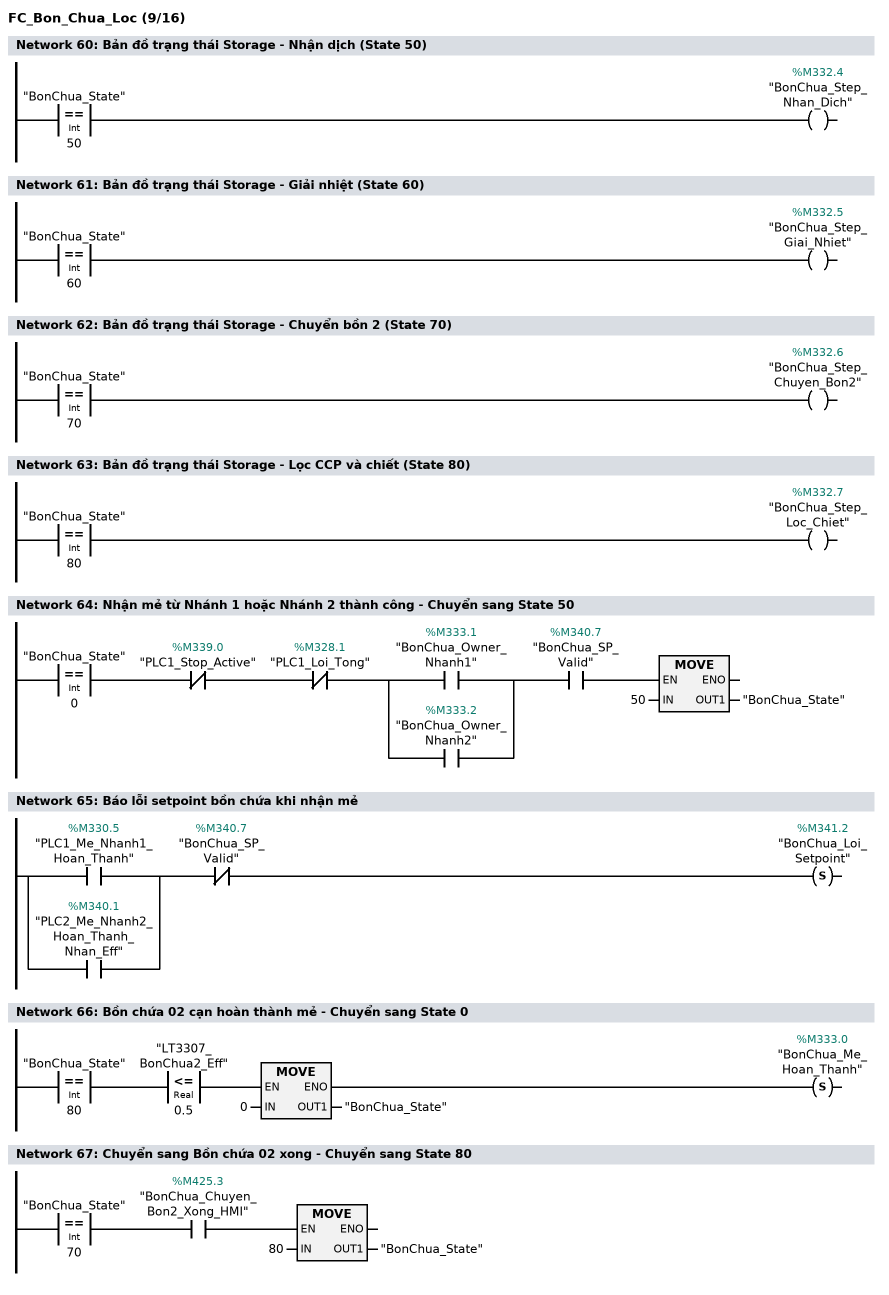
   RUNG wire#powerrail
      { S7_Templates := "SrcType := Int" } EQ_Contact(in1 := "BonChua_State", in2 := 50)
      Coil( "BonChua_Step_Nhan_Dich" )
   END_RUNG
   // the same network as SCL:
   "BonChua_Step_Nhan_Dich" := "BonChua_State" = 50;
END_REGION

REGION Network 61: Bản đồ trạng thái Storage - Giải nhiệt (State 60)
   RUNG wire#powerrail
      { S7_Templates := "SrcType := Int" } EQ_Contact(in1 := "BonChua_State", in2 := 60)
      Coil( "BonChua_Step_Giai_Nhiet" )
   END_RUNG
   // the same network as SCL:
   "BonChua_Step_Giai_Nhiet" := "BonChua_State" = 60;
END_REGION

REGION Network 62: Bản đồ trạng thái Storage - Chuyển bồn 2 (State 70)
   RUNG wire#powerrail
      { S7_Templates := "SrcType := Int" } EQ_Contact(in1 := "BonChua_State", in2 := 70)
      Coil( "BonChua_Step_Chuyen_Bon2" )
   END_RUNG
   // the same network as SCL:
   "BonChua_Step_Chuyen_Bon2" := "BonChua_State" = 70;
END_REGION

REGION Network 63: Bản đồ trạng thái Storage - Lọc CCP và chiết (State 80)
   RUNG wire#powerrail
      { S7_Templates := "SrcType := Int" } EQ_Contact(in1 := "BonChua_State", in2 := 80)
      Coil( "BonChua_Step_Loc_Chiet" )
   END_RUNG
   // the same network as SCL:
   "BonChua_Step_Loc_Chiet" := "BonChua_State" = 80;
END_REGION

REGION Network 64: Nhận mẻ từ Nhánh 1 hoặc Nhánh 2 thành công - Chuyển sang State 50
   RUNG wire#powerrail
      { S7_Templates := "SrcType := Int" } EQ_Contact(in1 := "BonChua_State", in2 := 0)
      I_Contact( "PLC1_Stop_Active" )
      I_Contact( "PLC1_Loi_Tong" )
      wire#w1
      Contact( "BonChua_Owner_Nhanh1" )
      wire#w2
      Contact( "BonChua_SP_Valid" )
      { S7_GenerateENO := "TRUE" } Move(in := 50, out1 => "BonChua_State")
   END_RUNG
   RUNG wire#w1
      Contact( "BonChua_Owner_Nhanh2" )
   END_RUNG wire#w2
   // the same network as SCL:
   IF ("BonChua_State" = 0) AND NOT "PLC1_Stop_Active" AND NOT "PLC1_Loi_Tong" AND ("BonChua_Owner_Nhanh1" OR "BonChua_Owner_Nhanh2") AND "BonChua_SP_Valid" THEN
       "BonChua_State" := 50;
   END_IF;
END_REGION

REGION Network 65: Báo lỗi setpoint bồn chứa khi nhận mẻ
   RUNG wire#powerrail
      Contact( "PLC1_Me_Nhanh1_Hoan_Thanh" )
      wire#w1
      I_Contact( "BonChua_SP_Valid" )
      S_Coil( "BonChua_Loi_Setpoint" )
   END_RUNG
   RUNG wire#powerrail
      Contact( "PLC2_Me_Nhanh2_Hoan_Thanh_Nhan_Eff" )
   END_RUNG wire#w1
   // the same network as SCL:
   IF ("PLC1_Me_Nhanh1_Hoan_Thanh" OR "PLC2_Me_Nhanh2_Hoan_Thanh_Nhan_Eff") AND NOT "BonChua_SP_Valid" THEN
       "BonChua_Loi_Setpoint" := TRUE;
   END_IF;
END_REGION

REGION Network 66: Bồn chứa 02 cạn hoàn thành mẻ - Chuyển sang State 0
   RUNG wire#powerrail
      { S7_Templates := "SrcType := Int" } EQ_Contact(in1 := "BonChua_State", in2 := 80)
      { S7_Templates := "SrcType := Real" } LE_Contact(in1 := "LT3307_BonChua2_Eff", in2 := 0.5)
      { S7_GenerateENO := "TRUE" } Move(in := 0, out1 => "BonChua_State")
      S_Coil( "BonChua_Me_Hoan_Thanh" )
   END_RUNG
   // the same network as SCL:
   // ENO of a box is taken as its EN; it also drops when the box reports an error
   #_w1 := ("BonChua_State" = 80) AND ("LT3307_BonChua2_Eff" <= 0.5);
   IF #_w1 THEN
       "BonChua_State" := 0;
       "BonChua_Me_Hoan_Thanh" := TRUE;
   END_IF;
END_REGION

REGION Network 67: Chuyển sang Bồn chứa 02 xong - Chuyển sang State 80
   RUNG wire#powerrail
      { S7_Templates := "SrcType := Int" } EQ_Contact(in1 := "BonChua_State", in2 := 70)
      Contact( "BonChua_Chuyen_Bon2_Xong_HMI" )
      { S7_GenerateENO := "TRUE" } Move(in := 80, out1 => "BonChua_State")
   END_RUNG
   // the same network as SCL:
   IF ("BonChua_State" = 70) AND "BonChua_Chuyen_Bon2_Xong_HMI" THEN "BonChua_State" := 80; END_IF;
END_REGION

REGION Network 68: Đạt 45 độ C chuyển Bồn chứa 02 - Chuyển sang State 70
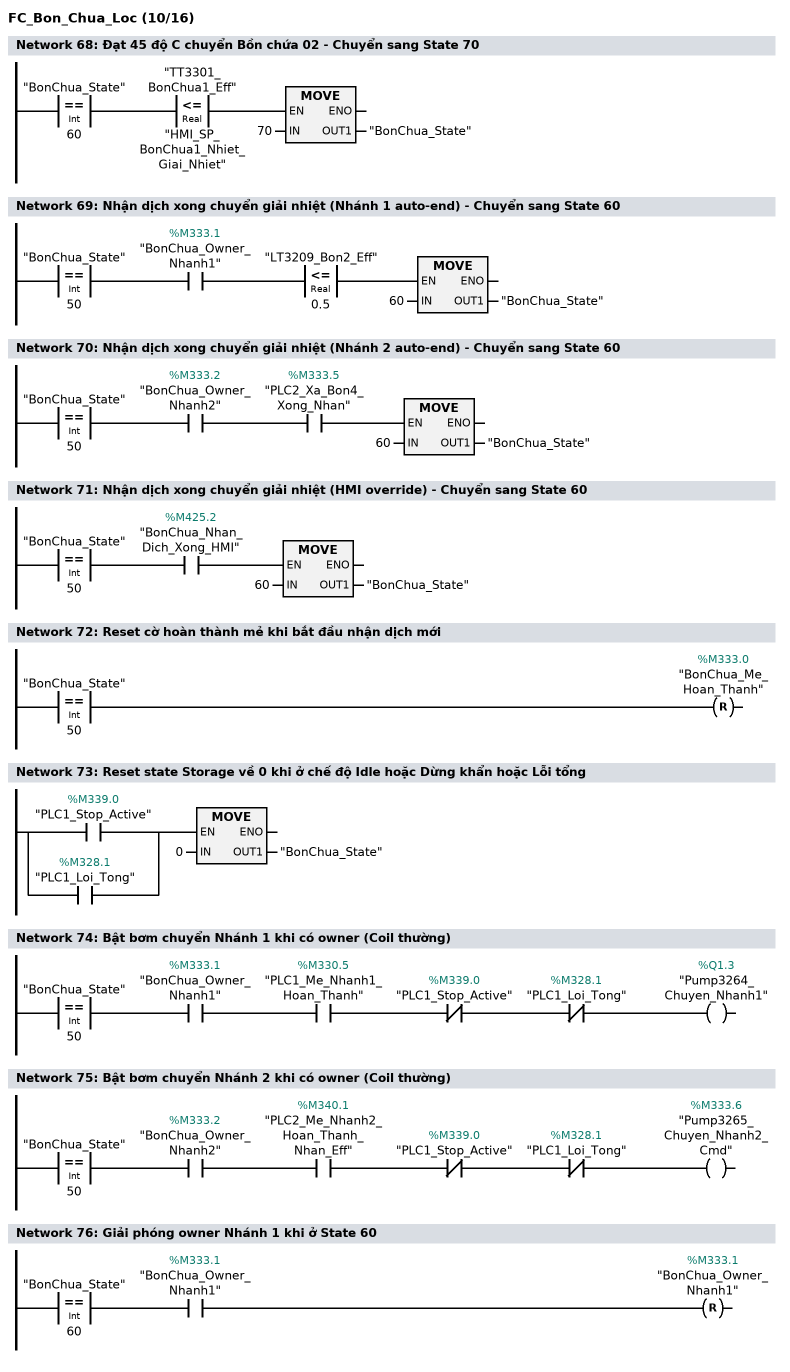
   RUNG wire#powerrail
      { S7_Templates := "SrcType := Int" } EQ_Contact(in1 := "BonChua_State", in2 := 60)
      { S7_Templates := "SrcType := Real" } LE_Contact(in1 := "TT3301_BonChua1_Eff", in2 := "HMI_SP_BonChua1_Nhiet_Giai_Nhiet")
      { S7_GenerateENO := "TRUE" } Move(in := 70, out1 => "BonChua_State")
   END_RUNG
   // the same network as SCL:
   IF ("BonChua_State" = 60) AND ("TT3301_BonChua1_Eff" <= "HMI_SP_BonChua1_Nhiet_Giai_Nhiet") THEN
       "BonChua_State" := 70;
   END_IF;
END_REGION

REGION Network 69: Nhận dịch xong chuyển giải nhiệt (Nhánh 1 auto-end) - Chuyển sang State 60
   RUNG wire#powerrail
      { S7_Templates := "SrcType := Int" } EQ_Contact(in1 := "BonChua_State", in2 := 50)
      Contact( "BonChua_Owner_Nhanh1" )
      { S7_Templates := "SrcType := Real" } LE_Contact(in1 := "LT3209_Bon2_Eff", in2 := 0.5)
      { S7_GenerateENO := "TRUE" } Move(in := 60, out1 => "BonChua_State")
   END_RUNG
   // the same network as SCL:
   IF ("BonChua_State" = 50) AND "BonChua_Owner_Nhanh1" AND ("LT3209_Bon2_Eff" <= 0.5) THEN
       "BonChua_State" := 60;
   END_IF;
END_REGION

REGION Network 70: Nhận dịch xong chuyển giải nhiệt (Nhánh 2 auto-end) - Chuyển sang State 60
   RUNG wire#powerrail
      { S7_Templates := "SrcType := Int" } EQ_Contact(in1 := "BonChua_State", in2 := 50)
      Contact( "BonChua_Owner_Nhanh2" )
      Contact( "PLC2_Xa_Bon4_Xong_Nhan" )
      { S7_GenerateENO := "TRUE" } Move(in := 60, out1 => "BonChua_State")
   END_RUNG
   // the same network as SCL:
   IF ("BonChua_State" = 50) AND "BonChua_Owner_Nhanh2" AND "PLC2_Xa_Bon4_Xong_Nhan" THEN
       "BonChua_State" := 60;
   END_IF;
END_REGION

REGION Network 71: Nhận dịch xong chuyển giải nhiệt (HMI override) - Chuyển sang State 60
   RUNG wire#powerrail
      { S7_Templates := "SrcType := Int" } EQ_Contact(in1 := "BonChua_State", in2 := 50)
      Contact( "BonChua_Nhan_Dich_Xong_HMI" )
      { S7_GenerateENO := "TRUE" } Move(in := 60, out1 => "BonChua_State")
   END_RUNG
   // the same network as SCL:
   IF ("BonChua_State" = 50) AND "BonChua_Nhan_Dich_Xong_HMI" THEN "BonChua_State" := 60; END_IF;
END_REGION

REGION Network 72: Reset cờ hoàn thành mẻ khi bắt đầu nhận dịch mới
   RUNG wire#powerrail
      { S7_Templates := "SrcType := Int" } EQ_Contact(in1 := "BonChua_State", in2 := 50)
      R_Coil( "BonChua_Me_Hoan_Thanh" )
   END_RUNG
   // the same network as SCL:
   IF "BonChua_State" = 50 THEN "BonChua_Me_Hoan_Thanh" := FALSE; END_IF;
END_REGION

REGION Network 73: Reset state Storage về 0 khi ở chế độ Idle hoặc Dừng khẩn hoặc Lỗi tổng
   RUNG wire#powerrail
      Contact( "PLC1_Stop_Active" )
      wire#w1
      { S7_GenerateENO := "TRUE" } Move(in := 0, out1 => "BonChua_State")
   END_RUNG
   RUNG wire#powerrail
      Contact( "PLC1_Loi_Tong" )
   END_RUNG wire#w1
   // the same network as SCL:
   IF "PLC1_Stop_Active" OR "PLC1_Loi_Tong" THEN "BonChua_State" := 0; END_IF;
END_REGION

REGION Network 74: Bật bơm chuyển Nhánh 1 khi có owner (Coil thường)
   RUNG wire#powerrail
      { S7_Templates := "SrcType := Int" } EQ_Contact(in1 := "BonChua_State", in2 := 50)
      Contact( "BonChua_Owner_Nhanh1" )
      Contact( "PLC1_Me_Nhanh1_Hoan_Thanh" )
      I_Contact( "PLC1_Stop_Active" )
      I_Contact( "PLC1_Loi_Tong" )
      Coil( "Pump3264_Chuyen_Nhanh1" )
   END_RUNG
   // the same network as SCL:
   "Pump3264_Chuyen_Nhanh1" := ("BonChua_State" = 50) AND "BonChua_Owner_Nhanh1" AND "PLC1_Me_Nhanh1_Hoan_Thanh" AND NOT "PLC1_Stop_Active" AND NOT "PLC1_Loi_Tong";
END_REGION

REGION Network 75: Bật bơm chuyển Nhánh 2 khi có owner (Coil thường)
   RUNG wire#powerrail
      { S7_Templates := "SrcType := Int" } EQ_Contact(in1 := "BonChua_State", in2 := 50)
      Contact( "BonChua_Owner_Nhanh2" )
      Contact( "PLC2_Me_Nhanh2_Hoan_Thanh_Nhan_Eff" )
      I_Contact( "PLC1_Stop_Active" )
      I_Contact( "PLC1_Loi_Tong" )
      Coil( "Pump3265_Chuyen_Nhanh2_Cmd" )
   END_RUNG
   // the same network as SCL:
   "Pump3265_Chuyen_Nhanh2_Cmd" := ("BonChua_State" = 50) AND "BonChua_Owner_Nhanh2" AND "PLC2_Me_Nhanh2_Hoan_Thanh_Nhan_Eff" AND NOT "PLC1_Stop_Active" AND NOT "PLC1_Loi_Tong";
END_REGION

REGION Network 76: Giải phóng owner Nhánh 1 khi ở State 60
   RUNG wire#powerrail
      { S7_Templates := "SrcType := Int" } EQ_Contact(in1 := "BonChua_State", in2 := 60)
      Contact( "BonChua_Owner_Nhanh1" )
      R_Coil( "BonChua_Owner_Nhanh1" )
   END_RUNG
   // the same network as SCL:
   IF ("BonChua_State" = 60) AND "BonChua_Owner_Nhanh1" THEN "BonChua_Owner_Nhanh1" := FALSE; END_IF;
END_REGION

REGION Network 77: Giải phóng owner Nhánh 2 khi ở State 60
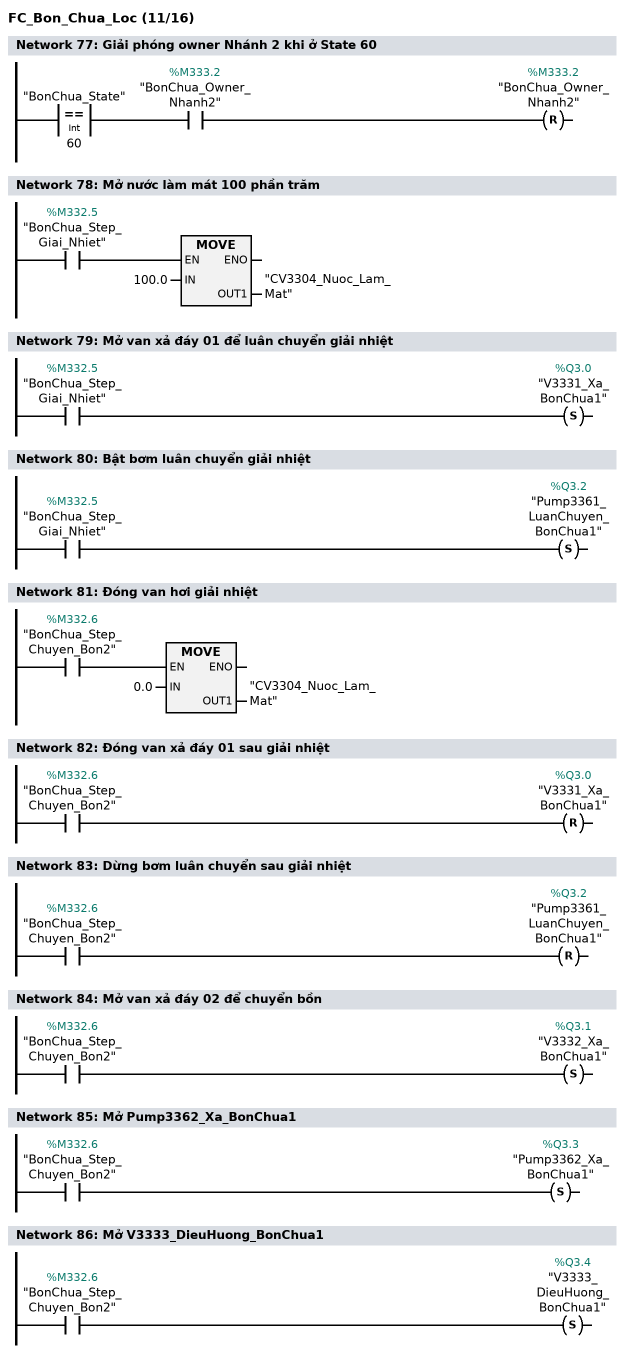
   RUNG wire#powerrail
      { S7_Templates := "SrcType := Int" } EQ_Contact(in1 := "BonChua_State", in2 := 60)
      Contact( "BonChua_Owner_Nhanh2" )
      R_Coil( "BonChua_Owner_Nhanh2" )
   END_RUNG
   // the same network as SCL:
   IF ("BonChua_State" = 60) AND "BonChua_Owner_Nhanh2" THEN "BonChua_Owner_Nhanh2" := FALSE; END_IF;
END_REGION

REGION Network 78: Mở nước làm mát 100 phần trăm
   RUNG wire#powerrail
      Contact( "BonChua_Step_Giai_Nhiet" )
      { S7_GenerateENO := "TRUE" } Move(in := 100.0, out1 => "CV3304_Nuoc_Lam_Mat")
   END_RUNG
   // the same network as SCL:
   IF "BonChua_Step_Giai_Nhiet" THEN "CV3304_Nuoc_Lam_Mat" := 100.0; END_IF;
END_REGION

REGION Network 79: Mở van xả đáy 01 để luân chuyển giải nhiệt
   RUNG wire#powerrail
      Contact( "BonChua_Step_Giai_Nhiet" )
      S_Coil( "V3331_Xa_BonChua1" )
   END_RUNG
   // the same network as SCL:
   IF "BonChua_Step_Giai_Nhiet" THEN "V3331_Xa_BonChua1" := TRUE; END_IF;
END_REGION

REGION Network 80: Bật bơm luân chuyển giải nhiệt
   RUNG wire#powerrail
      Contact( "BonChua_Step_Giai_Nhiet" )
      S_Coil( "Pump3361_LuanChuyen_BonChua1" )
   END_RUNG
   // the same network as SCL:
   IF "BonChua_Step_Giai_Nhiet" THEN "Pump3361_LuanChuyen_BonChua1" := TRUE; END_IF;
END_REGION

REGION Network 81: Đóng van hơi giải nhiệt
   RUNG wire#powerrail
      Contact( "BonChua_Step_Chuyen_Bon2" )
      { S7_GenerateENO := "TRUE" } Move(in := 0.0, out1 => "CV3304_Nuoc_Lam_Mat")
   END_RUNG
   // the same network as SCL:
   IF "BonChua_Step_Chuyen_Bon2" THEN "CV3304_Nuoc_Lam_Mat" := 0.0; END_IF;
END_REGION

REGION Network 82: Đóng van xả đáy 01 sau giải nhiệt
   RUNG wire#powerrail
      Contact( "BonChua_Step_Chuyen_Bon2" )
      R_Coil( "V3331_Xa_BonChua1" )
   END_RUNG
   // the same network as SCL:
   IF "BonChua_Step_Chuyen_Bon2" THEN "V3331_Xa_BonChua1" := FALSE; END_IF;
END_REGION

REGION Network 83: Dừng bơm luân chuyển sau giải nhiệt
   RUNG wire#powerrail
      Contact( "BonChua_Step_Chuyen_Bon2" )
      R_Coil( "Pump3361_LuanChuyen_BonChua1" )
   END_RUNG
   // the same network as SCL:
   IF "BonChua_Step_Chuyen_Bon2" THEN "Pump3361_LuanChuyen_BonChua1" := FALSE; END_IF;
END_REGION

REGION Network 84: Mở van xả đáy 02 để chuyển bồn
   RUNG wire#powerrail
      Contact( "BonChua_Step_Chuyen_Bon2" )
      S_Coil( "V3332_Xa_BonChua1" )
   END_RUNG
   // the same network as SCL:
   IF "BonChua_Step_Chuyen_Bon2" THEN "V3332_Xa_BonChua1" := TRUE; END_IF;
END_REGION

REGION Network 85: Mở Pump3362_Xa_BonChua1
   RUNG wire#powerrail
      Contact( "BonChua_Step_Chuyen_Bon2" )
      S_Coil( "Pump3362_Xa_BonChua1" )
   END_RUNG
   // the same network as SCL:
   IF "BonChua_Step_Chuyen_Bon2" THEN "Pump3362_Xa_BonChua1" := TRUE; END_IF;
END_REGION

REGION Network 86: Mở V3333_DieuHuong_BonChua1
   RUNG wire#powerrail
      Contact( "BonChua_Step_Chuyen_Bon2" )
      S_Coil( "V3333_DieuHuong_BonChua1" )
   END_RUNG
   // the same network as SCL:
   IF "BonChua_Step_Chuyen_Bon2" THEN "V3333_DieuHuong_BonChua1" := TRUE; END_IF;
END_REGION

REGION Network 87: Mở V3334_DieuHuong_BonChua1
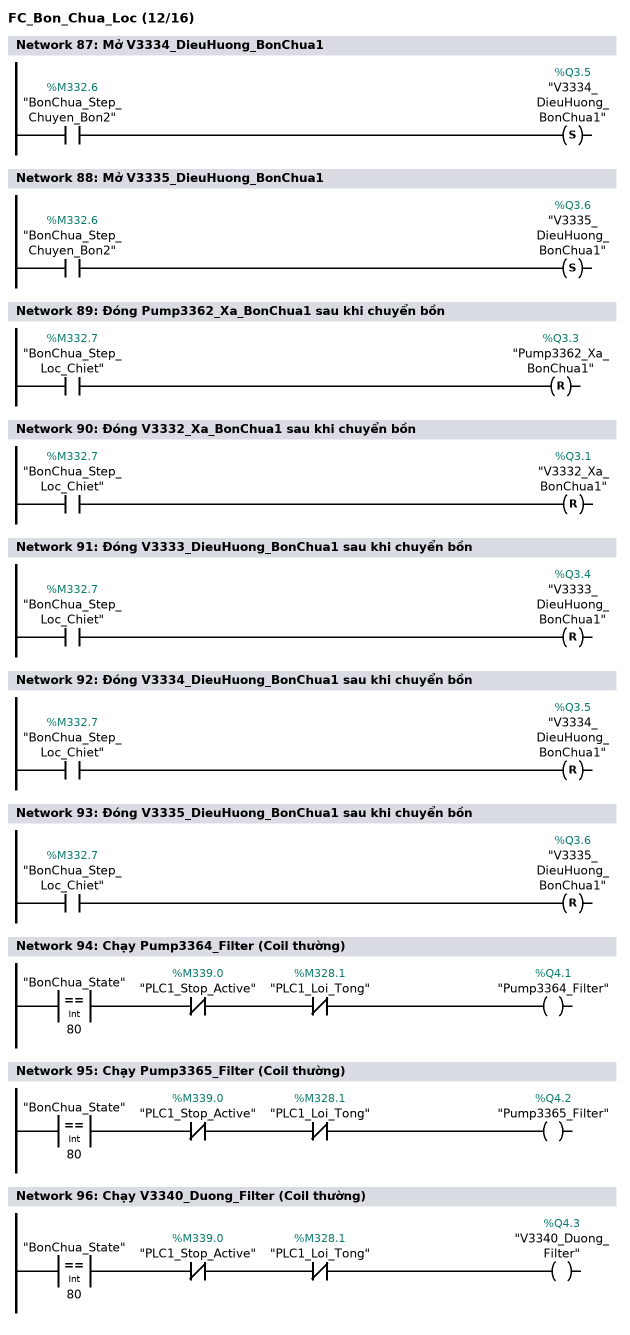
   RUNG wire#powerrail
      Contact( "BonChua_Step_Chuyen_Bon2" )
      S_Coil( "V3334_DieuHuong_BonChua1" )
   END_RUNG
   // the same network as SCL:
   IF "BonChua_Step_Chuyen_Bon2" THEN "V3334_DieuHuong_BonChua1" := TRUE; END_IF;
END_REGION

REGION Network 88: Mở V3335_DieuHuong_BonChua1
   RUNG wire#powerrail
      Contact( "BonChua_Step_Chuyen_Bon2" )
      S_Coil( "V3335_DieuHuong_BonChua1" )
   END_RUNG
   // the same network as SCL:
   IF "BonChua_Step_Chuyen_Bon2" THEN "V3335_DieuHuong_BonChua1" := TRUE; END_IF;
END_REGION

REGION Network 89: Đóng Pump3362_Xa_BonChua1 sau khi chuyển bồn
   RUNG wire#powerrail
      Contact( "BonChua_Step_Loc_Chiet" )
      R_Coil( "Pump3362_Xa_BonChua1" )
   END_RUNG
   // the same network as SCL:
   IF "BonChua_Step_Loc_Chiet" THEN "Pump3362_Xa_BonChua1" := FALSE; END_IF;
END_REGION

REGION Network 90: Đóng V3332_Xa_BonChua1 sau khi chuyển bồn
   RUNG wire#powerrail
      Contact( "BonChua_Step_Loc_Chiet" )
      R_Coil( "V3332_Xa_BonChua1" )
   END_RUNG
   // the same network as SCL:
   IF "BonChua_Step_Loc_Chiet" THEN "V3332_Xa_BonChua1" := FALSE; END_IF;
END_REGION

REGION Network 91: Đóng V3333_DieuHuong_BonChua1 sau khi chuyển bồn
   RUNG wire#powerrail
      Contact( "BonChua_Step_Loc_Chiet" )
      R_Coil( "V3333_DieuHuong_BonChua1" )
   END_RUNG
   // the same network as SCL:
   IF "BonChua_Step_Loc_Chiet" THEN "V3333_DieuHuong_BonChua1" := FALSE; END_IF;
END_REGION

REGION Network 92: Đóng V3334_DieuHuong_BonChua1 sau khi chuyển bồn
   RUNG wire#powerrail
      Contact( "BonChua_Step_Loc_Chiet" )
      R_Coil( "V3334_DieuHuong_BonChua1" )
   END_RUNG
   // the same network as SCL:
   IF "BonChua_Step_Loc_Chiet" THEN "V3334_DieuHuong_BonChua1" := FALSE; END_IF;
END_REGION

REGION Network 93: Đóng V3335_DieuHuong_BonChua1 sau khi chuyển bồn
   RUNG wire#powerrail
      Contact( "BonChua_Step_Loc_Chiet" )
      R_Coil( "V3335_DieuHuong_BonChua1" )
   END_RUNG
   // the same network as SCL:
   IF "BonChua_Step_Loc_Chiet" THEN "V3335_DieuHuong_BonChua1" := FALSE; END_IF;
END_REGION

REGION Network 94: Chạy Pump3364_Filter (Coil thường)
   RUNG wire#powerrail
      { S7_Templates := "SrcType := Int" } EQ_Contact(in1 := "BonChua_State", in2 := 80)
      I_Contact( "PLC1_Stop_Active" )
      I_Contact( "PLC1_Loi_Tong" )
      Coil( "Pump3364_Filter" )
   END_RUNG
   // the same network as SCL:
   "Pump3364_Filter" := ("BonChua_State" = 80) AND NOT "PLC1_Stop_Active" AND NOT "PLC1_Loi_Tong";
END_REGION

REGION Network 95: Chạy Pump3365_Filter (Coil thường)
   RUNG wire#powerrail
      { S7_Templates := "SrcType := Int" } EQ_Contact(in1 := "BonChua_State", in2 := 80)
      I_Contact( "PLC1_Stop_Active" )
      I_Contact( "PLC1_Loi_Tong" )
      Coil( "Pump3365_Filter" )
   END_RUNG
   // the same network as SCL:
   "Pump3365_Filter" := ("BonChua_State" = 80) AND NOT "PLC1_Stop_Active" AND NOT "PLC1_Loi_Tong";
END_REGION

REGION Network 96: Chạy V3340_Duong_Filter (Coil thường)
   RUNG wire#powerrail
      { S7_Templates := "SrcType := Int" } EQ_Contact(in1 := "BonChua_State", in2 := 80)
      I_Contact( "PLC1_Stop_Active" )
      I_Contact( "PLC1_Loi_Tong" )
      Coil( "V3340_Duong_Filter" )
   END_RUNG
   // the same network as SCL:
   "V3340_Duong_Filter" := ("BonChua_State" = 80) AND NOT "PLC1_Stop_Active" AND NOT "PLC1_Loi_Tong";
END_REGION

REGION Network 97: Chạy V3341_Duong_Filter (Coil thường)
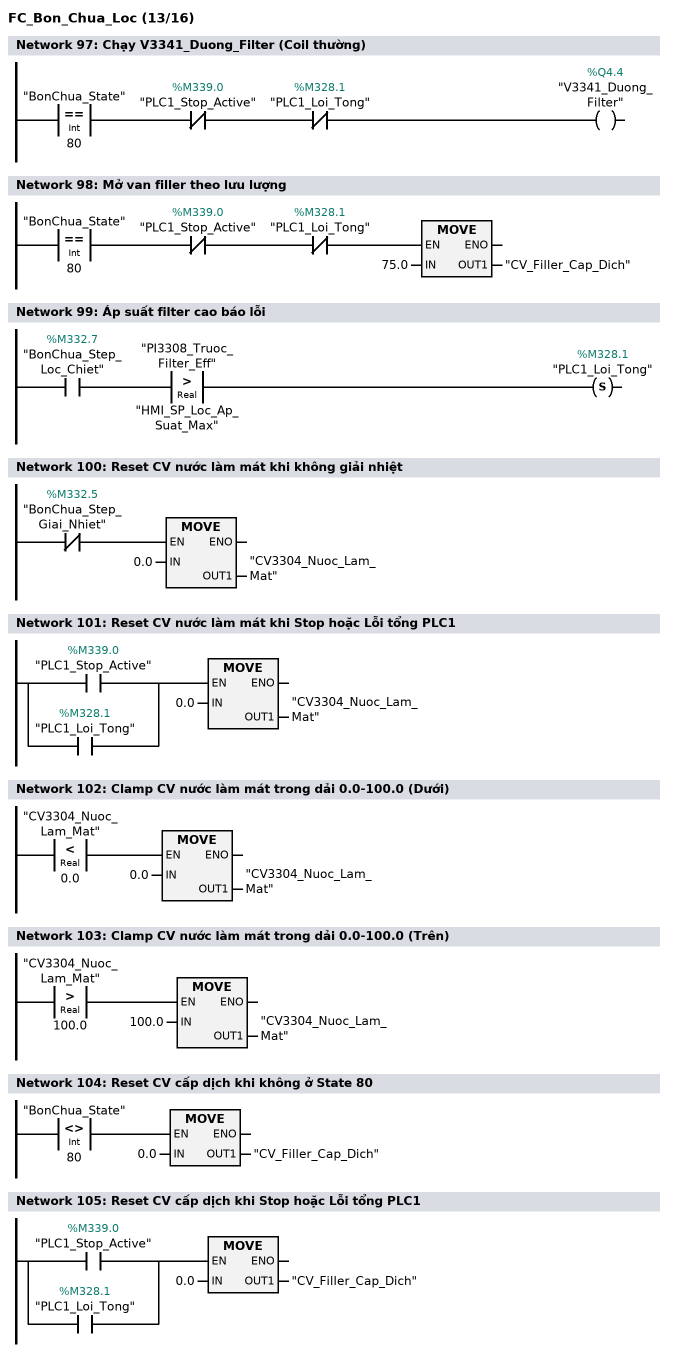
   RUNG wire#powerrail
      { S7_Templates := "SrcType := Int" } EQ_Contact(in1 := "BonChua_State", in2 := 80)
      I_Contact( "PLC1_Stop_Active" )
      I_Contact( "PLC1_Loi_Tong" )
      Coil( "V3341_Duong_Filter" )
   END_RUNG
   // the same network as SCL:
   "V3341_Duong_Filter" := ("BonChua_State" = 80) AND NOT "PLC1_Stop_Active" AND NOT "PLC1_Loi_Tong";
END_REGION

REGION Network 98: Mở van filler theo lưu lượng
   RUNG wire#powerrail
      { S7_Templates := "SrcType := Int" } EQ_Contact(in1 := "BonChua_State", in2 := 80)
      I_Contact( "PLC1_Stop_Active" )
      I_Contact( "PLC1_Loi_Tong" )
      { S7_GenerateENO := "TRUE" } Move(in := 75.0, out1 => "CV_Filler_Cap_Dich")
   END_RUNG
   // the same network as SCL:
   IF ("BonChua_State" = 80) AND NOT "PLC1_Stop_Active" AND NOT "PLC1_Loi_Tong" THEN
       "CV_Filler_Cap_Dich" := 75.0;
   END_IF;
END_REGION

REGION Network 99: Áp suất filter cao báo lỗi
   RUNG wire#powerrail
      Contact( "BonChua_Step_Loc_Chiet" )
      { S7_Templates := "SrcType := Real" } GT_Contact(in1 := "PI3308_Truoc_Filter_Eff", in2 := "HMI_SP_Loc_Ap_Suat_Max")
      S_Coil( "PLC1_Loi_Tong" )
   END_RUNG
   // the same network as SCL:
   IF "BonChua_Step_Loc_Chiet" AND ("PI3308_Truoc_Filter_Eff" > "HMI_SP_Loc_Ap_Suat_Max") THEN
       "PLC1_Loi_Tong" := TRUE;
   END_IF;
END_REGION

REGION Network 100: Reset CV nước làm mát khi không giải nhiệt
   RUNG wire#powerrail
      I_Contact( "BonChua_Step_Giai_Nhiet" )
      { S7_GenerateENO := "TRUE" } Move(in := 0.0, out1 => "CV3304_Nuoc_Lam_Mat")
   END_RUNG
   // the same network as SCL:
   IF NOT "BonChua_Step_Giai_Nhiet" THEN "CV3304_Nuoc_Lam_Mat" := 0.0; END_IF;
END_REGION

REGION Network 101: Reset CV nước làm mát khi Stop hoặc Lỗi tổng PLC1
   RUNG wire#powerrail
      Contact( "PLC1_Stop_Active" )
      wire#w1
      { S7_GenerateENO := "TRUE" } Move(in := 0.0, out1 => "CV3304_Nuoc_Lam_Mat")
   END_RUNG
   RUNG wire#powerrail
      Contact( "PLC1_Loi_Tong" )
   END_RUNG wire#w1
   // the same network as SCL:
   IF "PLC1_Stop_Active" OR "PLC1_Loi_Tong" THEN "CV3304_Nuoc_Lam_Mat" := 0.0; END_IF;
END_REGION

REGION Network 102: Clamp CV nước làm mát trong dải 0.0-100.0 (Dưới)
   RUNG wire#powerrail
      { S7_Templates := "SrcType := Real" } LT_Contact(in1 := "CV3304_Nuoc_Lam_Mat", in2 := 0.0)
      { S7_GenerateENO := "TRUE" } Move(in := 0.0, out1 => "CV3304_Nuoc_Lam_Mat")
   END_RUNG
   // the same network as SCL:
   IF "CV3304_Nuoc_Lam_Mat" < 0.0 THEN "CV3304_Nuoc_Lam_Mat" := 0.0; END_IF;
END_REGION

REGION Network 103: Clamp CV nước làm mát trong dải 0.0-100.0 (Trên)
   RUNG wire#powerrail
      { S7_Templates := "SrcType := Real" } GT_Contact(in1 := "CV3304_Nuoc_Lam_Mat", in2 := 100.0)
      { S7_GenerateENO := "TRUE" } Move(in := 100.0, out1 => "CV3304_Nuoc_Lam_Mat")
   END_RUNG
   // the same network as SCL:
   IF "CV3304_Nuoc_Lam_Mat" > 100.0 THEN "CV3304_Nuoc_Lam_Mat" := 100.0; END_IF;
END_REGION

REGION Network 104: Reset CV cấp dịch khi không ở State 80
   RUNG wire#powerrail
      { S7_Templates := "SrcType := Int" } NE_Contact(in1 := "BonChua_State", in2 := 80)
      { S7_GenerateENO := "TRUE" } Move(in := 0.0, out1 => "CV_Filler_Cap_Dich")
   END_RUNG
   // the same network as SCL:
   IF "BonChua_State" <> 80 THEN "CV_Filler_Cap_Dich" := 0.0; END_IF;
END_REGION

REGION Network 105: Reset CV cấp dịch khi Stop hoặc Lỗi tổng PLC1
   RUNG wire#powerrail
      Contact( "PLC1_Stop_Active" )
      wire#w1
      { S7_GenerateENO := "TRUE" } Move(in := 0.0, out1 => "CV_Filler_Cap_Dich")
   END_RUNG
   RUNG wire#powerrail
      Contact( "PLC1_Loi_Tong" )
   END_RUNG wire#w1
   // the same network as SCL:
   IF "PLC1_Stop_Active" OR "PLC1_Loi_Tong" THEN "CV_Filler_Cap_Dich" := 0.0; END_IF;
END_REGION

REGION Network 106: Clamp CV cấp dịch trong dải 0.0-100.0 (Dưới)
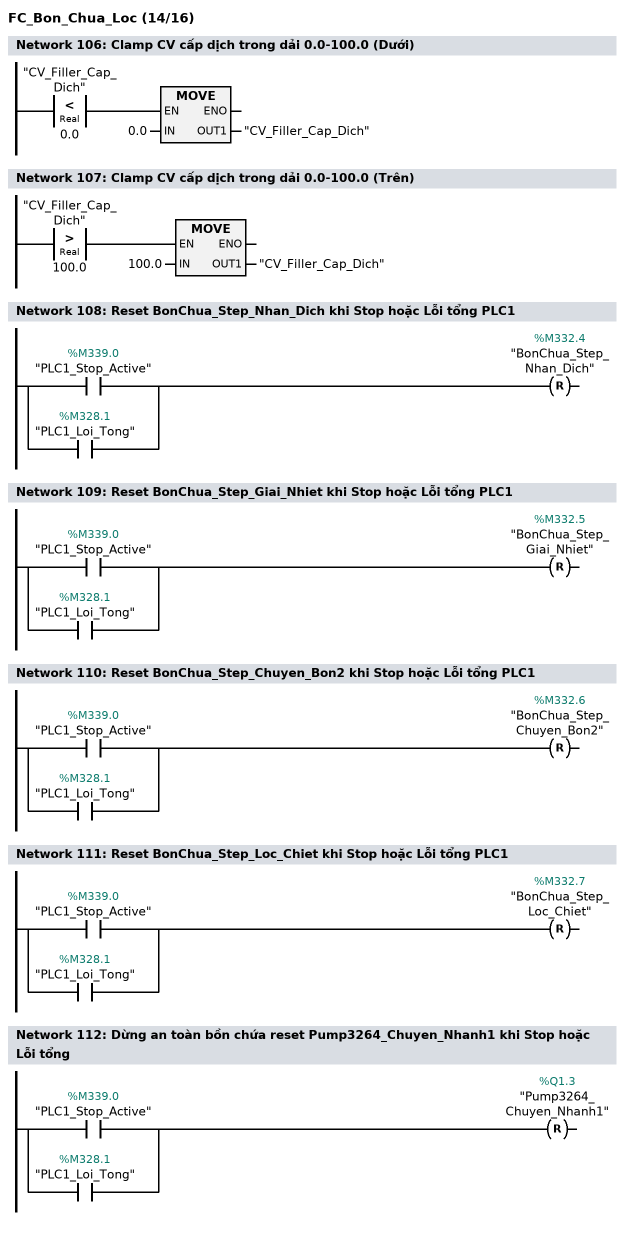
   RUNG wire#powerrail
      { S7_Templates := "SrcType := Real" } LT_Contact(in1 := "CV_Filler_Cap_Dich", in2 := 0.0)
      { S7_GenerateENO := "TRUE" } Move(in := 0.0, out1 => "CV_Filler_Cap_Dich")
   END_RUNG
   // the same network as SCL:
   IF "CV_Filler_Cap_Dich" < 0.0 THEN "CV_Filler_Cap_Dich" := 0.0; END_IF;
END_REGION

REGION Network 107: Clamp CV cấp dịch trong dải 0.0-100.0 (Trên)
   RUNG wire#powerrail
      { S7_Templates := "SrcType := Real" } GT_Contact(in1 := "CV_Filler_Cap_Dich", in2 := 100.0)
      { S7_GenerateENO := "TRUE" } Move(in := 100.0, out1 => "CV_Filler_Cap_Dich")
   END_RUNG
   // the same network as SCL:
   IF "CV_Filler_Cap_Dich" > 100.0 THEN "CV_Filler_Cap_Dich" := 100.0; END_IF;
END_REGION

REGION Network 108: Reset BonChua_Step_Nhan_Dich khi Stop hoặc Lỗi tổng PLC1
   RUNG wire#powerrail
      Contact( "PLC1_Stop_Active" )
      wire#w1
      R_Coil( "BonChua_Step_Nhan_Dich" )
   END_RUNG
   RUNG wire#powerrail
      Contact( "PLC1_Loi_Tong" )
   END_RUNG wire#w1
   // the same network as SCL:
   IF "PLC1_Stop_Active" OR "PLC1_Loi_Tong" THEN "BonChua_Step_Nhan_Dich" := FALSE; END_IF;
END_REGION

REGION Network 109: Reset BonChua_Step_Giai_Nhiet khi Stop hoặc Lỗi tổng PLC1
   RUNG wire#powerrail
      Contact( "PLC1_Stop_Active" )
      wire#w1
      R_Coil( "BonChua_Step_Giai_Nhiet" )
   END_RUNG
   RUNG wire#powerrail
      Contact( "PLC1_Loi_Tong" )
   END_RUNG wire#w1
   // the same network as SCL:
   IF "PLC1_Stop_Active" OR "PLC1_Loi_Tong" THEN "BonChua_Step_Giai_Nhiet" := FALSE; END_IF;
END_REGION

REGION Network 110: Reset BonChua_Step_Chuyen_Bon2 khi Stop hoặc Lỗi tổng PLC1
   RUNG wire#powerrail
      Contact( "PLC1_Stop_Active" )
      wire#w1
      R_Coil( "BonChua_Step_Chuyen_Bon2" )
   END_RUNG
   RUNG wire#powerrail
      Contact( "PLC1_Loi_Tong" )
   END_RUNG wire#w1
   // the same network as SCL:
   IF "PLC1_Stop_Active" OR "PLC1_Loi_Tong" THEN "BonChua_Step_Chuyen_Bon2" := FALSE; END_IF;
END_REGION

REGION Network 111: Reset BonChua_Step_Loc_Chiet khi Stop hoặc Lỗi tổng PLC1
   RUNG wire#powerrail
      Contact( "PLC1_Stop_Active" )
      wire#w1
      R_Coil( "BonChua_Step_Loc_Chiet" )
   END_RUNG
   RUNG wire#powerrail
      Contact( "PLC1_Loi_Tong" )
   END_RUNG wire#w1
   // the same network as SCL:
   IF "PLC1_Stop_Active" OR "PLC1_Loi_Tong" THEN "BonChua_Step_Loc_Chiet" := FALSE; END_IF;
END_REGION

REGION Network 112: Dừng an toàn bồn chứa reset Pump3264_Chuyen_Nhanh1 khi Stop hoặc Lỗi tổng
   RUNG wire#powerrail
      Contact( "PLC1_Stop_Active" )
      wire#w1
      R_Coil( "Pump3264_Chuyen_Nhanh1" )
   END_RUNG
   RUNG wire#powerrail
      Contact( "PLC1_Loi_Tong" )
   END_RUNG wire#w1
   // the same network as SCL:
   IF "PLC1_Stop_Active" OR "PLC1_Loi_Tong" THEN "Pump3264_Chuyen_Nhanh1" := FALSE; END_IF;
END_REGION

REGION Network 113: Dừng an toàn bồn chứa reset Pump3265_Chuyen_Nhanh2_Cmd khi Stop hoặc Lỗi tổng
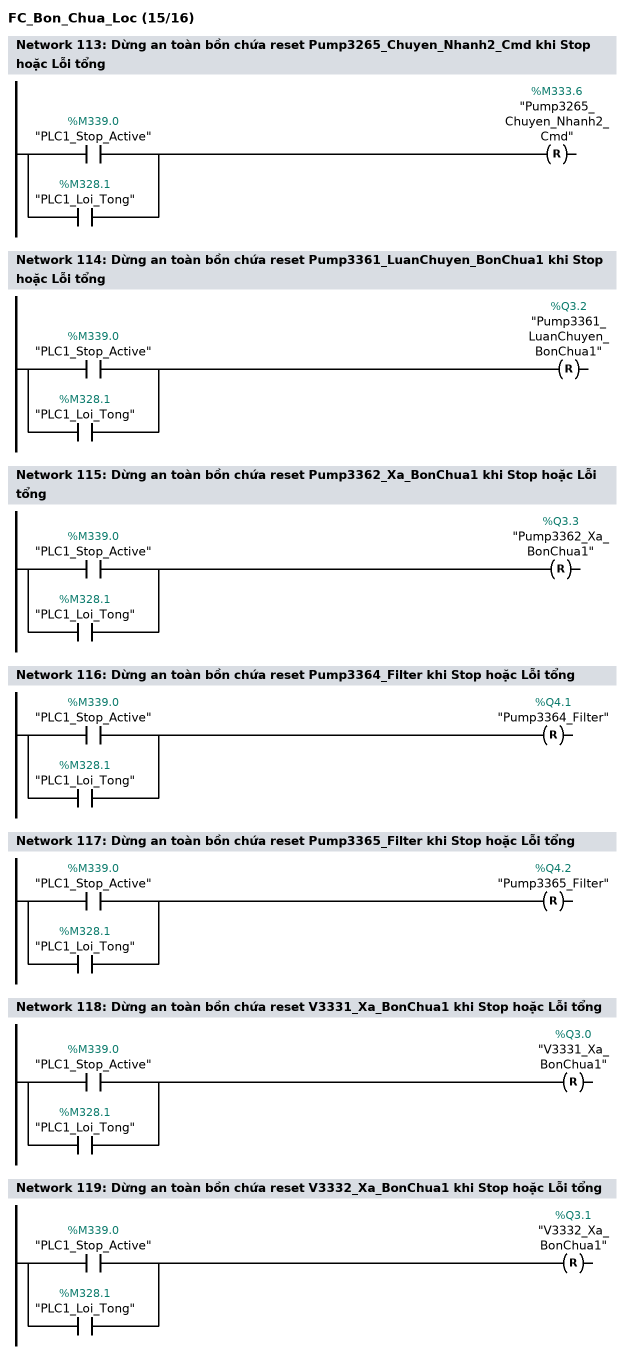
   RUNG wire#powerrail
      Contact( "PLC1_Stop_Active" )
      wire#w1
      R_Coil( "Pump3265_Chuyen_Nhanh2_Cmd" )
   END_RUNG
   RUNG wire#powerrail
      Contact( "PLC1_Loi_Tong" )
   END_RUNG wire#w1
   // the same network as SCL:
   IF "PLC1_Stop_Active" OR "PLC1_Loi_Tong" THEN "Pump3265_Chuyen_Nhanh2_Cmd" := FALSE; END_IF;
END_REGION

REGION Network 114: Dừng an toàn bồn chứa reset Pump3361_LuanChuyen_BonChua1 khi Stop hoặc Lỗi tổng
   RUNG wire#powerrail
      Contact( "PLC1_Stop_Active" )
      wire#w1
      R_Coil( "Pump3361_LuanChuyen_BonChua1" )
   END_RUNG
   RUNG wire#powerrail
      Contact( "PLC1_Loi_Tong" )
   END_RUNG wire#w1
   // the same network as SCL:
   IF "PLC1_Stop_Active" OR "PLC1_Loi_Tong" THEN "Pump3361_LuanChuyen_BonChua1" := FALSE; END_IF;
END_REGION

REGION Network 115: Dừng an toàn bồn chứa reset Pump3362_Xa_BonChua1 khi Stop hoặc Lỗi tổng
   RUNG wire#powerrail
      Contact( "PLC1_Stop_Active" )
      wire#w1
      R_Coil( "Pump3362_Xa_BonChua1" )
   END_RUNG
   RUNG wire#powerrail
      Contact( "PLC1_Loi_Tong" )
   END_RUNG wire#w1
   // the same network as SCL:
   IF "PLC1_Stop_Active" OR "PLC1_Loi_Tong" THEN "Pump3362_Xa_BonChua1" := FALSE; END_IF;
END_REGION

REGION Network 116: Dừng an toàn bồn chứa reset Pump3364_Filter khi Stop hoặc Lỗi tổng
   RUNG wire#powerrail
      Contact( "PLC1_Stop_Active" )
      wire#w1
      R_Coil( "Pump3364_Filter" )
   END_RUNG
   RUNG wire#powerrail
      Contact( "PLC1_Loi_Tong" )
   END_RUNG wire#w1
   // the same network as SCL:
   IF "PLC1_Stop_Active" OR "PLC1_Loi_Tong" THEN "Pump3364_Filter" := FALSE; END_IF;
END_REGION

REGION Network 117: Dừng an toàn bồn chứa reset Pump3365_Filter khi Stop hoặc Lỗi tổng
   RUNG wire#powerrail
      Contact( "PLC1_Stop_Active" )
      wire#w1
      R_Coil( "Pump3365_Filter" )
   END_RUNG
   RUNG wire#powerrail
      Contact( "PLC1_Loi_Tong" )
   END_RUNG wire#w1
   // the same network as SCL:
   IF "PLC1_Stop_Active" OR "PLC1_Loi_Tong" THEN "Pump3365_Filter" := FALSE; END_IF;
END_REGION

REGION Network 118: Dừng an toàn bồn chứa reset V3331_Xa_BonChua1 khi Stop hoặc Lỗi tổng
   RUNG wire#powerrail
      Contact( "PLC1_Stop_Active" )
      wire#w1
      R_Coil( "V3331_Xa_BonChua1" )
   END_RUNG
   RUNG wire#powerrail
      Contact( "PLC1_Loi_Tong" )
   END_RUNG wire#w1
   // the same network as SCL:
   IF "PLC1_Stop_Active" OR "PLC1_Loi_Tong" THEN "V3331_Xa_BonChua1" := FALSE; END_IF;
END_REGION

REGION Network 119: Dừng an toàn bồn chứa reset V3332_Xa_BonChua1 khi Stop hoặc Lỗi tổng
   RUNG wire#powerrail
      Contact( "PLC1_Stop_Active" )
      wire#w1
      R_Coil( "V3332_Xa_BonChua1" )
   END_RUNG
   RUNG wire#powerrail
      Contact( "PLC1_Loi_Tong" )
   END_RUNG wire#w1
   // the same network as SCL:
   IF "PLC1_Stop_Active" OR "PLC1_Loi_Tong" THEN "V3332_Xa_BonChua1" := FALSE; END_IF;
END_REGION

REGION Network 120: Dừng an toàn bồn chứa reset V3333_DieuHuong_BonChua1 khi Stop hoặc Lỗi tổng
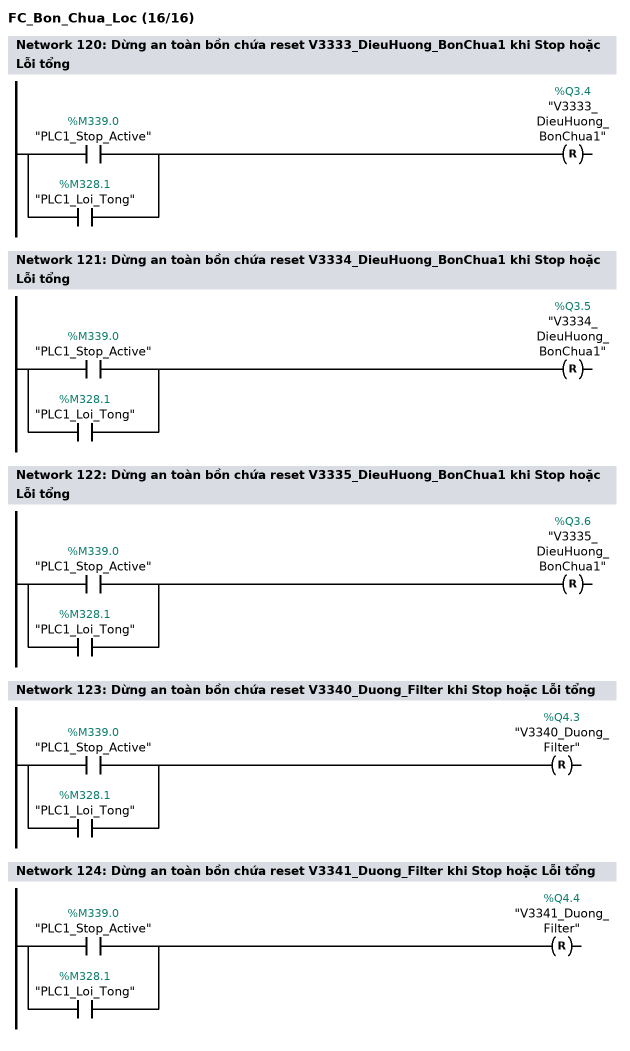
   RUNG wire#powerrail
      Contact( "PLC1_Stop_Active" )
      wire#w1
      R_Coil( "V3333_DieuHuong_BonChua1" )
   END_RUNG
   RUNG wire#powerrail
      Contact( "PLC1_Loi_Tong" )
   END_RUNG wire#w1
   // the same network as SCL:
   IF "PLC1_Stop_Active" OR "PLC1_Loi_Tong" THEN "V3333_DieuHuong_BonChua1" := FALSE; END_IF;
END_REGION

REGION Network 121: Dừng an toàn bồn chứa reset V3334_DieuHuong_BonChua1 khi Stop hoặc Lỗi tổng
   RUNG wire#powerrail
      Contact( "PLC1_Stop_Active" )
      wire#w1
      R_Coil( "V3334_DieuHuong_BonChua1" )
   END_RUNG
   RUNG wire#powerrail
      Contact( "PLC1_Loi_Tong" )
   END_RUNG wire#w1
   // the same network as SCL:
   IF "PLC1_Stop_Active" OR "PLC1_Loi_Tong" THEN "V3334_DieuHuong_BonChua1" := FALSE; END_IF;
END_REGION

REGION Network 122: Dừng an toàn bồn chứa reset V3335_DieuHuong_BonChua1 khi Stop hoặc Lỗi tổng
   RUNG wire#powerrail
      Contact( "PLC1_Stop_Active" )
      wire#w1
      R_Coil( "V3335_DieuHuong_BonChua1" )
   END_RUNG
   RUNG wire#powerrail
      Contact( "PLC1_Loi_Tong" )
   END_RUNG wire#w1
   // the same network as SCL:
   IF "PLC1_Stop_Active" OR "PLC1_Loi_Tong" THEN "V3335_DieuHuong_BonChua1" := FALSE; END_IF;
END_REGION

REGION Network 123: Dừng an toàn bồn chứa reset V3340_Duong_Filter khi Stop hoặc Lỗi tổng
   RUNG wire#powerrail
      Contact( "PLC1_Stop_Active" )
      wire#w1
      R_Coil( "V3340_Duong_Filter" )
   END_RUNG
   RUNG wire#powerrail
      Contact( "PLC1_Loi_Tong" )
   END_RUNG wire#w1
   // the same network as SCL:
   IF "PLC1_Stop_Active" OR "PLC1_Loi_Tong" THEN "V3340_Duong_Filter" := FALSE; END_IF;
END_REGION

REGION Network 124: Dừng an toàn bồn chứa reset V3341_Duong_Filter khi Stop hoặc Lỗi tổng
   RUNG wire#powerrail
      Contact( "PLC1_Stop_Active" )
      wire#w1
      R_Coil( "V3341_Duong_Filter" )
   END_RUNG
   RUNG wire#powerrail
      Contact( "PLC1_Loi_Tong" )
   END_RUNG wire#w1
   // the same network as SCL:
   IF "PLC1_Stop_Active" OR "PLC1_Loi_Tong" THEN "V3341_Duong_Filter" := FALSE; END_IF;
END_REGION
END_FUNCTION

FUNCTION "FC_HMI_Mirror_PLC1" : Void   // FC40, LAD
{ S7_Optimized_Access := 'TRUE' }
VERSION : 0.1
// stored: AutoNumber true, IsIECCheckEnabled false, SetENOAutomatically false, UDAEnableTagReadback false
BEGIN

REGION Network 1: Mirror V3230_Nuoc_Bon1
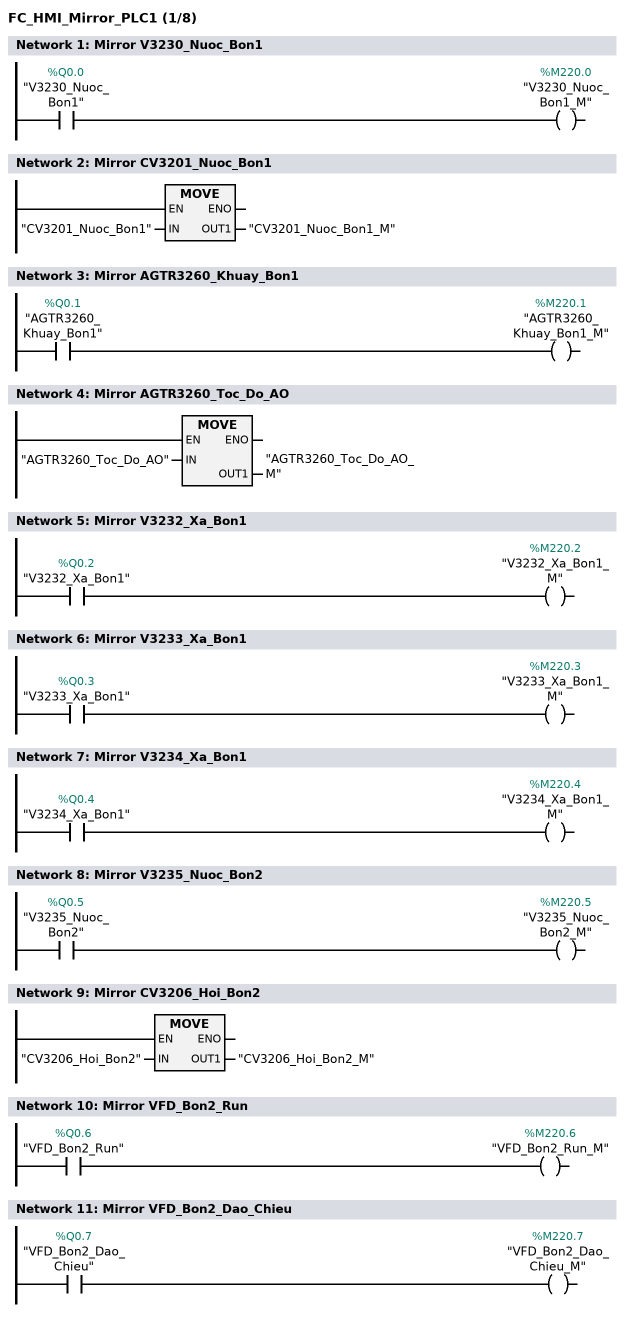
   RUNG wire#powerrail
      Contact( "V3230_Nuoc_Bon1" )
      Coil( "V3230_Nuoc_Bon1_M" )
   END_RUNG
   // the same network as SCL:
   "V3230_Nuoc_Bon1_M" := "V3230_Nuoc_Bon1";
END_REGION

REGION Network 2: Mirror CV3201_Nuoc_Bon1
   RUNG wire#powerrail
      { S7_GenerateENO := "TRUE" } Move(in := "CV3201_Nuoc_Bon1", out1 => "CV3201_Nuoc_Bon1_M")
   END_RUNG
   // the same network as SCL:
   "CV3201_Nuoc_Bon1_M" := "CV3201_Nuoc_Bon1";
END_REGION

REGION Network 3: Mirror AGTR3260_Khuay_Bon1
   RUNG wire#powerrail
      Contact( "AGTR3260_Khuay_Bon1" )
      Coil( "AGTR3260_Khuay_Bon1_M" )
   END_RUNG
   // the same network as SCL:
   "AGTR3260_Khuay_Bon1_M" := "AGTR3260_Khuay_Bon1";
END_REGION

REGION Network 4: Mirror AGTR3260_Toc_Do_AO
   RUNG wire#powerrail
      { S7_GenerateENO := "TRUE" } Move(in := "AGTR3260_Toc_Do_AO", out1 => "AGTR3260_Toc_Do_AO_M")
   END_RUNG
   // the same network as SCL:
   "AGTR3260_Toc_Do_AO_M" := "AGTR3260_Toc_Do_AO";
END_REGION

REGION Network 5: Mirror V3232_Xa_Bon1
   RUNG wire#powerrail
      Contact( "V3232_Xa_Bon1" )
      Coil( "V3232_Xa_Bon1_M" )
   END_RUNG
   // the same network as SCL:
   "V3232_Xa_Bon1_M" := "V3232_Xa_Bon1";
END_REGION

REGION Network 6: Mirror V3233_Xa_Bon1
   RUNG wire#powerrail
      Contact( "V3233_Xa_Bon1" )
      Coil( "V3233_Xa_Bon1_M" )
   END_RUNG
   // the same network as SCL:
   "V3233_Xa_Bon1_M" := "V3233_Xa_Bon1";
END_REGION

REGION Network 7: Mirror V3234_Xa_Bon1
   RUNG wire#powerrail
      Contact( "V3234_Xa_Bon1" )
      Coil( "V3234_Xa_Bon1_M" )
   END_RUNG
   // the same network as SCL:
   "V3234_Xa_Bon1_M" := "V3234_Xa_Bon1";
END_REGION

REGION Network 8: Mirror V3235_Nuoc_Bon2
   RUNG wire#powerrail
      Contact( "V3235_Nuoc_Bon2" )
      Coil( "V3235_Nuoc_Bon2_M" )
   END_RUNG
   // the same network as SCL:
   "V3235_Nuoc_Bon2_M" := "V3235_Nuoc_Bon2";
END_REGION

REGION Network 9: Mirror CV3206_Hoi_Bon2
   RUNG wire#powerrail
      { S7_GenerateENO := "TRUE" } Move(in := "CV3206_Hoi_Bon2", out1 => "CV3206_Hoi_Bon2_M")
   END_RUNG
   // the same network as SCL:
   "CV3206_Hoi_Bon2_M" := "CV3206_Hoi_Bon2";
END_REGION

REGION Network 10: Mirror VFD_Bon2_Run
   RUNG wire#powerrail
      Contact( "VFD_Bon2_Run" )
      Coil( "VFD_Bon2_Run_M" )
   END_RUNG
   // the same network as SCL:
   "VFD_Bon2_Run_M" := "VFD_Bon2_Run";
END_REGION

REGION Network 11: Mirror VFD_Bon2_Dao_Chieu
   RUNG wire#powerrail
      Contact( "VFD_Bon2_Dao_Chieu" )
      Coil( "VFD_Bon2_Dao_Chieu_M" )
   END_RUNG
   // the same network as SCL:
   "VFD_Bon2_Dao_Chieu_M" := "VFD_Bon2_Dao_Chieu";
END_REGION

REGION Network 12: Mirror VFD_Bon2_Toc_Do_AO
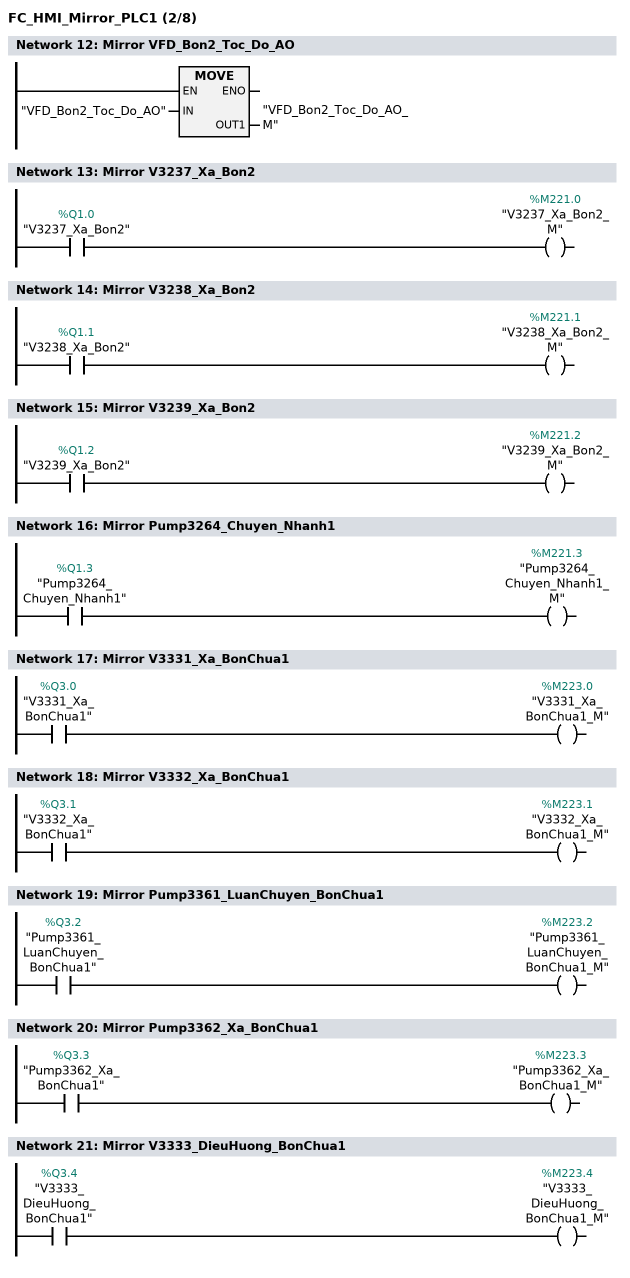
   RUNG wire#powerrail
      { S7_GenerateENO := "TRUE" } Move(in := "VFD_Bon2_Toc_Do_AO", out1 => "VFD_Bon2_Toc_Do_AO_M")
   END_RUNG
   // the same network as SCL:
   "VFD_Bon2_Toc_Do_AO_M" := "VFD_Bon2_Toc_Do_AO";
END_REGION

REGION Network 13: Mirror V3237_Xa_Bon2
   RUNG wire#powerrail
      Contact( "V3237_Xa_Bon2" )
      Coil( "V3237_Xa_Bon2_M" )
   END_RUNG
   // the same network as SCL:
   "V3237_Xa_Bon2_M" := "V3237_Xa_Bon2";
END_REGION

REGION Network 14: Mirror V3238_Xa_Bon2
   RUNG wire#powerrail
      Contact( "V3238_Xa_Bon2" )
      Coil( "V3238_Xa_Bon2_M" )
   END_RUNG
   // the same network as SCL:
   "V3238_Xa_Bon2_M" := "V3238_Xa_Bon2";
END_REGION

REGION Network 15: Mirror V3239_Xa_Bon2
   RUNG wire#powerrail
      Contact( "V3239_Xa_Bon2" )
      Coil( "V3239_Xa_Bon2_M" )
   END_RUNG
   // the same network as SCL:
   "V3239_Xa_Bon2_M" := "V3239_Xa_Bon2";
END_REGION

REGION Network 16: Mirror Pump3264_Chuyen_Nhanh1
   RUNG wire#powerrail
      Contact( "Pump3264_Chuyen_Nhanh1" )
      Coil( "Pump3264_Chuyen_Nhanh1_M" )
   END_RUNG
   // the same network as SCL:
   "Pump3264_Chuyen_Nhanh1_M" := "Pump3264_Chuyen_Nhanh1";
END_REGION

REGION Network 17: Mirror V3331_Xa_BonChua1
   RUNG wire#powerrail
      Contact( "V3331_Xa_BonChua1" )
      Coil( "V3331_Xa_BonChua1_M" )
   END_RUNG
   // the same network as SCL:
   "V3331_Xa_BonChua1_M" := "V3331_Xa_BonChua1";
END_REGION

REGION Network 18: Mirror V3332_Xa_BonChua1
   RUNG wire#powerrail
      Contact( "V3332_Xa_BonChua1" )
      Coil( "V3332_Xa_BonChua1_M" )
   END_RUNG
   // the same network as SCL:
   "V3332_Xa_BonChua1_M" := "V3332_Xa_BonChua1";
END_REGION

REGION Network 19: Mirror Pump3361_LuanChuyen_BonChua1
   RUNG wire#powerrail
      Contact( "Pump3361_LuanChuyen_BonChua1" )
      Coil( "Pump3361_LuanChuyen_BonChua1_M" )
   END_RUNG
   // the same network as SCL:
   "Pump3361_LuanChuyen_BonChua1_M" := "Pump3361_LuanChuyen_BonChua1";
END_REGION

REGION Network 20: Mirror Pump3362_Xa_BonChua1
   RUNG wire#powerrail
      Contact( "Pump3362_Xa_BonChua1" )
      Coil( "Pump3362_Xa_BonChua1_M" )
   END_RUNG
   // the same network as SCL:
   "Pump3362_Xa_BonChua1_M" := "Pump3362_Xa_BonChua1";
END_REGION

REGION Network 21: Mirror V3333_DieuHuong_BonChua1
   RUNG wire#powerrail
      Contact( "V3333_DieuHuong_BonChua1" )
      Coil( "V3333_DieuHuong_BonChua1_M" )
   END_RUNG
   // the same network as SCL:
   "V3333_DieuHuong_BonChua1_M" := "V3333_DieuHuong_BonChua1";
END_REGION

REGION Network 22: Mirror V3334_DieuHuong_BonChua1
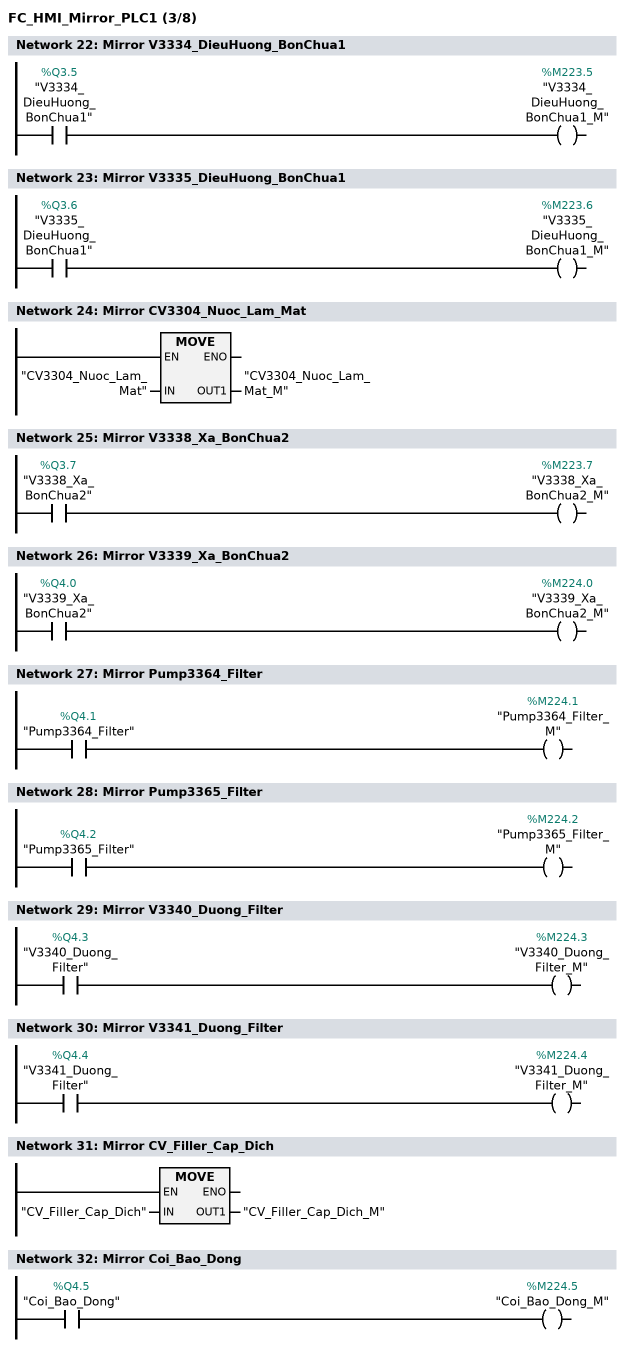
   RUNG wire#powerrail
      Contact( "V3334_DieuHuong_BonChua1" )
      Coil( "V3334_DieuHuong_BonChua1_M" )
   END_RUNG
   // the same network as SCL:
   "V3334_DieuHuong_BonChua1_M" := "V3334_DieuHuong_BonChua1";
END_REGION

REGION Network 23: Mirror V3335_DieuHuong_BonChua1
   RUNG wire#powerrail
      Contact( "V3335_DieuHuong_BonChua1" )
      Coil( "V3335_DieuHuong_BonChua1_M" )
   END_RUNG
   // the same network as SCL:
   "V3335_DieuHuong_BonChua1_M" := "V3335_DieuHuong_BonChua1";
END_REGION

REGION Network 24: Mirror CV3304_Nuoc_Lam_Mat
   RUNG wire#powerrail
      { S7_GenerateENO := "TRUE" } Move(in := "CV3304_Nuoc_Lam_Mat", out1 => "CV3304_Nuoc_Lam_Mat_M")
   END_RUNG
   // the same network as SCL:
   "CV3304_Nuoc_Lam_Mat_M" := "CV3304_Nuoc_Lam_Mat";
END_REGION

REGION Network 25: Mirror V3338_Xa_BonChua2
   RUNG wire#powerrail
      Contact( "V3338_Xa_BonChua2" )
      Coil( "V3338_Xa_BonChua2_M" )
   END_RUNG
   // the same network as SCL:
   "V3338_Xa_BonChua2_M" := "V3338_Xa_BonChua2";
END_REGION

REGION Network 26: Mirror V3339_Xa_BonChua2
   RUNG wire#powerrail
      Contact( "V3339_Xa_BonChua2" )
      Coil( "V3339_Xa_BonChua2_M" )
   END_RUNG
   // the same network as SCL:
   "V3339_Xa_BonChua2_M" := "V3339_Xa_BonChua2";
END_REGION

REGION Network 27: Mirror Pump3364_Filter
   RUNG wire#powerrail
      Contact( "Pump3364_Filter" )
      Coil( "Pump3364_Filter_M" )
   END_RUNG
   // the same network as SCL:
   "Pump3364_Filter_M" := "Pump3364_Filter";
END_REGION

REGION Network 28: Mirror Pump3365_Filter
   RUNG wire#powerrail
      Contact( "Pump3365_Filter" )
      Coil( "Pump3365_Filter_M" )
   END_RUNG
   // the same network as SCL:
   "Pump3365_Filter_M" := "Pump3365_Filter";
END_REGION

REGION Network 29: Mirror V3340_Duong_Filter
   RUNG wire#powerrail
      Contact( "V3340_Duong_Filter" )
      Coil( "V3340_Duong_Filter_M" )
   END_RUNG
   // the same network as SCL:
   "V3340_Duong_Filter_M" := "V3340_Duong_Filter";
END_REGION

REGION Network 30: Mirror V3341_Duong_Filter
   RUNG wire#powerrail
      Contact( "V3341_Duong_Filter" )
      Coil( "V3341_Duong_Filter_M" )
   END_RUNG
   // the same network as SCL:
   "V3341_Duong_Filter_M" := "V3341_Duong_Filter";
END_REGION

REGION Network 31: Mirror CV_Filler_Cap_Dich
   RUNG wire#powerrail
      { S7_GenerateENO := "TRUE" } Move(in := "CV_Filler_Cap_Dich", out1 => "CV_Filler_Cap_Dich_M")
   END_RUNG
   // the same network as SCL:
   "CV_Filler_Cap_Dich_M" := "CV_Filler_Cap_Dich";
END_REGION

REGION Network 32: Mirror Coi_Bao_Dong
   RUNG wire#powerrail
      Contact( "Coi_Bao_Dong" )
      Coil( "Coi_Bao_Dong_M" )
   END_RUNG
   // the same network as SCL:
   "Coi_Bao_Dong_M" := "Coi_Bao_Dong";
END_REGION

REGION Network 33: Mirror Pump3265_Chuyen_Nhanh2_Cmd
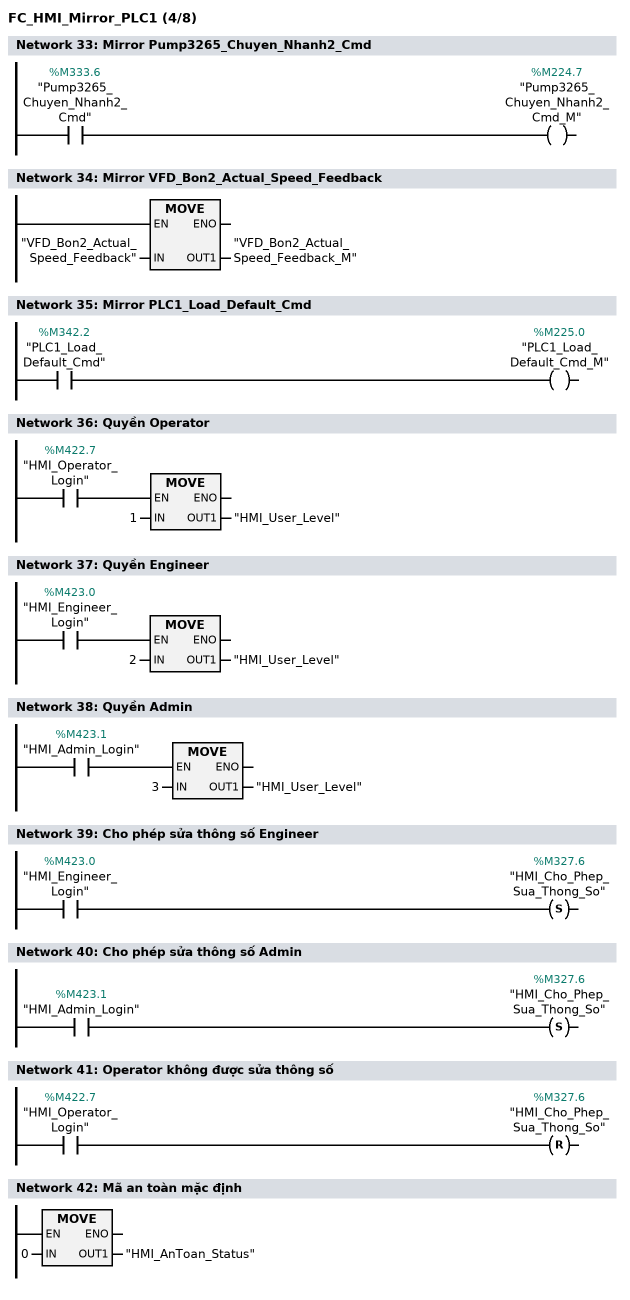
   RUNG wire#powerrail
      Contact( "Pump3265_Chuyen_Nhanh2_Cmd" )
      Coil( "Pump3265_Chuyen_Nhanh2_Cmd_M" )
   END_RUNG
   // the same network as SCL:
   "Pump3265_Chuyen_Nhanh2_Cmd_M" := "Pump3265_Chuyen_Nhanh2_Cmd";
END_REGION

REGION Network 34: Mirror VFD_Bon2_Actual_Speed_Feedback
   RUNG wire#powerrail
      { S7_GenerateENO := "TRUE" } Move(in := "VFD_Bon2_Actual_Speed_Feedback", out1 => "VFD_Bon2_Actual_Speed_Feedback_M")
   END_RUNG
   // the same network as SCL:
   "VFD_Bon2_Actual_Speed_Feedback_M" := "VFD_Bon2_Actual_Speed_Feedback";
END_REGION

REGION Network 35: Mirror PLC1_Load_Default_Cmd
   RUNG wire#powerrail
      Contact( "PLC1_Load_Default_Cmd" )
      Coil( "PLC1_Load_Default_Cmd_M" )
   END_RUNG
   // the same network as SCL:
   "PLC1_Load_Default_Cmd_M" := "PLC1_Load_Default_Cmd";
END_REGION

REGION Network 36: Quyền Operator
   RUNG wire#powerrail
      Contact( "HMI_Operator_Login" )
      { S7_GenerateENO := "TRUE" } Move(in := 1, out1 => "HMI_User_Level")
   END_RUNG
   // the same network as SCL:
   IF "HMI_Operator_Login" THEN "HMI_User_Level" := 1; END_IF;
END_REGION

REGION Network 37: Quyền Engineer
   RUNG wire#powerrail
      Contact( "HMI_Engineer_Login" )
      { S7_GenerateENO := "TRUE" } Move(in := 2, out1 => "HMI_User_Level")
   END_RUNG
   // the same network as SCL:
   IF "HMI_Engineer_Login" THEN "HMI_User_Level" := 2; END_IF;
END_REGION

REGION Network 38: Quyền Admin
   RUNG wire#powerrail
      Contact( "HMI_Admin_Login" )
      { S7_GenerateENO := "TRUE" } Move(in := 3, out1 => "HMI_User_Level")
   END_RUNG
   // the same network as SCL:
   IF "HMI_Admin_Login" THEN "HMI_User_Level" := 3; END_IF;
END_REGION

REGION Network 39: Cho phép sửa thông số Engineer
   RUNG wire#powerrail
      Contact( "HMI_Engineer_Login" )
      S_Coil( "HMI_Cho_Phep_Sua_Thong_So" )
   END_RUNG
   // the same network as SCL:
   IF "HMI_Engineer_Login" THEN "HMI_Cho_Phep_Sua_Thong_So" := TRUE; END_IF;
END_REGION

REGION Network 40: Cho phép sửa thông số Admin
   RUNG wire#powerrail
      Contact( "HMI_Admin_Login" )
      S_Coil( "HMI_Cho_Phep_Sua_Thong_So" )
   END_RUNG
   // the same network as SCL:
   IF "HMI_Admin_Login" THEN "HMI_Cho_Phep_Sua_Thong_So" := TRUE; END_IF;
END_REGION

REGION Network 41: Operator không được sửa thông số
   RUNG wire#powerrail
      Contact( "HMI_Operator_Login" )
      R_Coil( "HMI_Cho_Phep_Sua_Thong_So" )
   END_RUNG
   // the same network as SCL:
   IF "HMI_Operator_Login" THEN "HMI_Cho_Phep_Sua_Thong_So" := FALSE; END_IF;
END_REGION

REGION Network 42: Mã an toàn mặc định
   RUNG wire#powerrail
      { S7_GenerateENO := "TRUE" } Move(in := 0, out1 => "HMI_AnToan_Status")
   END_RUNG
   // the same network as SCL:
   "HMI_AnToan_Status" := 0;
END_REGION

REGION Network 43: Mã cảnh báo dosing PLC1
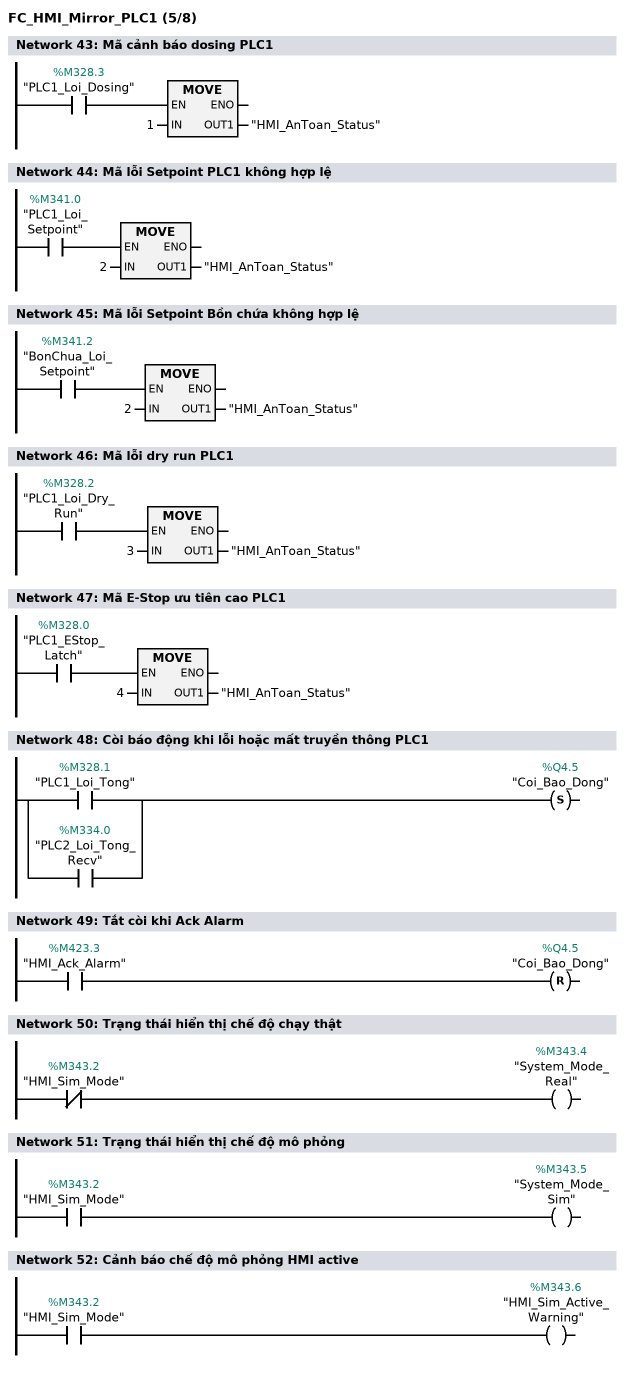
   RUNG wire#powerrail
      Contact( "PLC1_Loi_Dosing" )
      { S7_GenerateENO := "TRUE" } Move(in := 1, out1 => "HMI_AnToan_Status")
   END_RUNG
   // the same network as SCL:
   IF "PLC1_Loi_Dosing" THEN "HMI_AnToan_Status" := 1; END_IF;
END_REGION

REGION Network 44: Mã lỗi Setpoint PLC1 không hợp lệ
   RUNG wire#powerrail
      Contact( "PLC1_Loi_Setpoint" )
      { S7_GenerateENO := "TRUE" } Move(in := 2, out1 => "HMI_AnToan_Status")
   END_RUNG
   // the same network as SCL:
   IF "PLC1_Loi_Setpoint" THEN "HMI_AnToan_Status" := 2; END_IF;
END_REGION

REGION Network 45: Mã lỗi Setpoint Bồn chứa không hợp lệ
   RUNG wire#powerrail
      Contact( "BonChua_Loi_Setpoint" )
      { S7_GenerateENO := "TRUE" } Move(in := 2, out1 => "HMI_AnToan_Status")
   END_RUNG
   // the same network as SCL:
   IF "BonChua_Loi_Setpoint" THEN "HMI_AnToan_Status" := 2; END_IF;
END_REGION

REGION Network 46: Mã lỗi dry run PLC1
   RUNG wire#powerrail
      Contact( "PLC1_Loi_Dry_Run" )
      { S7_GenerateENO := "TRUE" } Move(in := 3, out1 => "HMI_AnToan_Status")
   END_RUNG
   // the same network as SCL:
   IF "PLC1_Loi_Dry_Run" THEN "HMI_AnToan_Status" := 3; END_IF;
END_REGION

REGION Network 47: Mã E-Stop ưu tiên cao PLC1
   RUNG wire#powerrail
      Contact( "PLC1_EStop_Latch" )
      { S7_GenerateENO := "TRUE" } Move(in := 4, out1 => "HMI_AnToan_Status")
   END_RUNG
   // the same network as SCL:
   IF "PLC1_EStop_Latch" THEN "HMI_AnToan_Status" := 4; END_IF;
END_REGION

REGION Network 48: Còi báo động khi lỗi hoặc mất truyền thông PLC1
   RUNG wire#powerrail
      Contact( "PLC1_Loi_Tong" )
      wire#w1
      S_Coil( "Coi_Bao_Dong" )
   END_RUNG
   RUNG wire#powerrail
      Contact( "PLC2_Loi_Tong_Recv" )
   END_RUNG wire#w1
   // the same network as SCL:
   IF "PLC1_Loi_Tong" OR "PLC2_Loi_Tong_Recv" THEN "Coi_Bao_Dong" := TRUE; END_IF;
END_REGION

REGION Network 49: Tắt còi khi Ack Alarm
   RUNG wire#powerrail
      Contact( "HMI_Ack_Alarm" )
      R_Coil( "Coi_Bao_Dong" )
   END_RUNG
   // the same network as SCL:
   IF "HMI_Ack_Alarm" THEN "Coi_Bao_Dong" := FALSE; END_IF;
END_REGION

REGION Network 50: Trạng thái hiển thị chế độ chạy thật
   RUNG wire#powerrail
      I_Contact( "HMI_Sim_Mode" )
      Coil( "System_Mode_Real" )
   END_RUNG
   // the same network as SCL:
   "System_Mode_Real" := NOT "HMI_Sim_Mode";
END_REGION

REGION Network 51: Trạng thái hiển thị chế độ mô phỏng
   RUNG wire#powerrail
      Contact( "HMI_Sim_Mode" )
      Coil( "System_Mode_Sim" )
   END_RUNG
   // the same network as SCL:
   "System_Mode_Sim" := "HMI_Sim_Mode";
END_REGION

REGION Network 52: Cảnh báo chế độ mô phỏng HMI active
   RUNG wire#powerrail
      Contact( "HMI_Sim_Mode" )
      Coil( "HMI_Sim_Active_Warning" )
   END_RUNG
   // the same network as SCL:
   "HMI_Sim_Active_Warning" := "HMI_Sim_Mode";
END_REGION

REGION Network 53: Reset LS3202_Bon1_Cao_HMI khi ở chế độ chạy thật
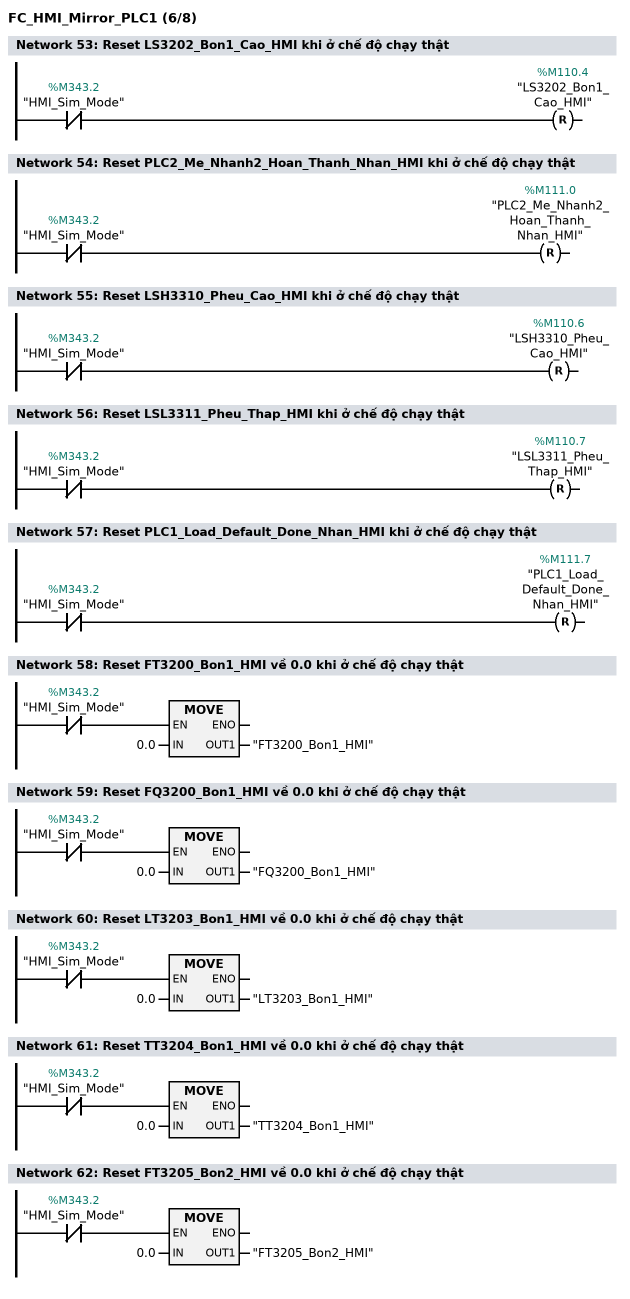
   RUNG wire#powerrail
      I_Contact( "HMI_Sim_Mode" )
      R_Coil( "LS3202_Bon1_Cao_HMI" )
   END_RUNG
   // the same network as SCL:
   IF NOT "HMI_Sim_Mode" THEN "LS3202_Bon1_Cao_HMI" := FALSE; END_IF;
END_REGION

REGION Network 54: Reset PLC2_Me_Nhanh2_Hoan_Thanh_Nhan_HMI khi ở chế độ chạy thật
   RUNG wire#powerrail
      I_Contact( "HMI_Sim_Mode" )
      R_Coil( "PLC2_Me_Nhanh2_Hoan_Thanh_Nhan_HMI" )
   END_RUNG
   // the same network as SCL:
   IF NOT "HMI_Sim_Mode" THEN "PLC2_Me_Nhanh2_Hoan_Thanh_Nhan_HMI" := FALSE; END_IF;
END_REGION

REGION Network 55: Reset LSH3310_Pheu_Cao_HMI khi ở chế độ chạy thật
   RUNG wire#powerrail
      I_Contact( "HMI_Sim_Mode" )
      R_Coil( "LSH3310_Pheu_Cao_HMI" )
   END_RUNG
   // the same network as SCL:
   IF NOT "HMI_Sim_Mode" THEN "LSH3310_Pheu_Cao_HMI" := FALSE; END_IF;
END_REGION

REGION Network 56: Reset LSL3311_Pheu_Thap_HMI khi ở chế độ chạy thật
   RUNG wire#powerrail
      I_Contact( "HMI_Sim_Mode" )
      R_Coil( "LSL3311_Pheu_Thap_HMI" )
   END_RUNG
   // the same network as SCL:
   IF NOT "HMI_Sim_Mode" THEN "LSL3311_Pheu_Thap_HMI" := FALSE; END_IF;
END_REGION

REGION Network 57: Reset PLC1_Load_Default_Done_Nhan_HMI khi ở chế độ chạy thật
   RUNG wire#powerrail
      I_Contact( "HMI_Sim_Mode" )
      R_Coil( "PLC1_Load_Default_Done_Nhan_HMI" )
   END_RUNG
   // the same network as SCL:
   IF NOT "HMI_Sim_Mode" THEN "PLC1_Load_Default_Done_Nhan_HMI" := FALSE; END_IF;
END_REGION

REGION Network 58: Reset FT3200_Bon1_HMI về 0.0 khi ở chế độ chạy thật
   RUNG wire#powerrail
      I_Contact( "HMI_Sim_Mode" )
      { S7_GenerateENO := "TRUE" } Move(in := 0.0, out1 => "FT3200_Bon1_HMI")
   END_RUNG
   // the same network as SCL:
   IF NOT "HMI_Sim_Mode" THEN "FT3200_Bon1_HMI" := 0.0; END_IF;
END_REGION

REGION Network 59: Reset FQ3200_Bon1_HMI về 0.0 khi ở chế độ chạy thật
   RUNG wire#powerrail
      I_Contact( "HMI_Sim_Mode" )
      { S7_GenerateENO := "TRUE" } Move(in := 0.0, out1 => "FQ3200_Bon1_HMI")
   END_RUNG
   // the same network as SCL:
   IF NOT "HMI_Sim_Mode" THEN "FQ3200_Bon1_HMI" := 0.0; END_IF;
END_REGION

REGION Network 60: Reset LT3203_Bon1_HMI về 0.0 khi ở chế độ chạy thật
   RUNG wire#powerrail
      I_Contact( "HMI_Sim_Mode" )
      { S7_GenerateENO := "TRUE" } Move(in := 0.0, out1 => "LT3203_Bon1_HMI")
   END_RUNG
   // the same network as SCL:
   IF NOT "HMI_Sim_Mode" THEN "LT3203_Bon1_HMI" := 0.0; END_IF;
END_REGION

REGION Network 61: Reset TT3204_Bon1_HMI về 0.0 khi ở chế độ chạy thật
   RUNG wire#powerrail
      I_Contact( "HMI_Sim_Mode" )
      { S7_GenerateENO := "TRUE" } Move(in := 0.0, out1 => "TT3204_Bon1_HMI")
   END_RUNG
   // the same network as SCL:
   IF NOT "HMI_Sim_Mode" THEN "TT3204_Bon1_HMI" := 0.0; END_IF;
END_REGION

REGION Network 62: Reset FT3205_Bon2_HMI về 0.0 khi ở chế độ chạy thật
   RUNG wire#powerrail
      I_Contact( "HMI_Sim_Mode" )
      { S7_GenerateENO := "TRUE" } Move(in := 0.0, out1 => "FT3205_Bon2_HMI")
   END_RUNG
   // the same network as SCL:
   IF NOT "HMI_Sim_Mode" THEN "FT3205_Bon2_HMI" := 0.0; END_IF;
END_REGION

REGION Network 63: Reset FQ3205_Bon2_HMI về 0.0 khi ở chế độ chạy thật
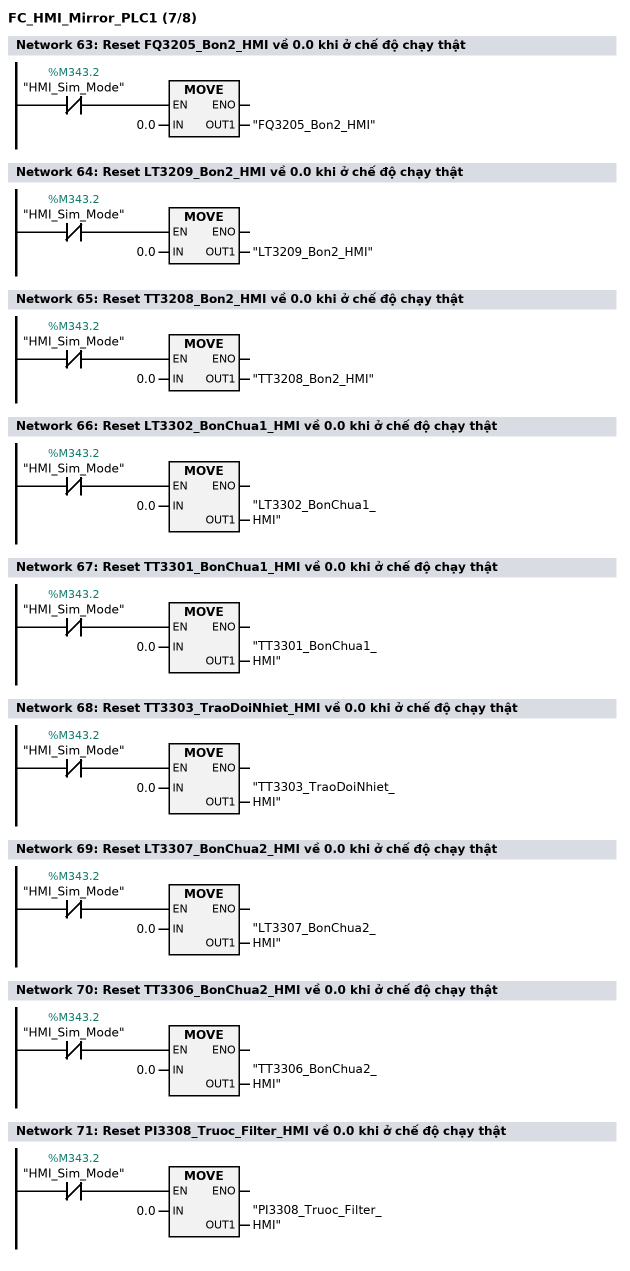
   RUNG wire#powerrail
      I_Contact( "HMI_Sim_Mode" )
      { S7_GenerateENO := "TRUE" } Move(in := 0.0, out1 => "FQ3205_Bon2_HMI")
   END_RUNG
   // the same network as SCL:
   IF NOT "HMI_Sim_Mode" THEN "FQ3205_Bon2_HMI" := 0.0; END_IF;
END_REGION

REGION Network 64: Reset LT3209_Bon2_HMI về 0.0 khi ở chế độ chạy thật
   RUNG wire#powerrail
      I_Contact( "HMI_Sim_Mode" )
      { S7_GenerateENO := "TRUE" } Move(in := 0.0, out1 => "LT3209_Bon2_HMI")
   END_RUNG
   // the same network as SCL:
   IF NOT "HMI_Sim_Mode" THEN "LT3209_Bon2_HMI" := 0.0; END_IF;
END_REGION

REGION Network 65: Reset TT3208_Bon2_HMI về 0.0 khi ở chế độ chạy thật
   RUNG wire#powerrail
      I_Contact( "HMI_Sim_Mode" )
      { S7_GenerateENO := "TRUE" } Move(in := 0.0, out1 => "TT3208_Bon2_HMI")
   END_RUNG
   // the same network as SCL:
   IF NOT "HMI_Sim_Mode" THEN "TT3208_Bon2_HMI" := 0.0; END_IF;
END_REGION

REGION Network 66: Reset LT3302_BonChua1_HMI về 0.0 khi ở chế độ chạy thật
   RUNG wire#powerrail
      I_Contact( "HMI_Sim_Mode" )
      { S7_GenerateENO := "TRUE" } Move(in := 0.0, out1 => "LT3302_BonChua1_HMI")
   END_RUNG
   // the same network as SCL:
   IF NOT "HMI_Sim_Mode" THEN "LT3302_BonChua1_HMI" := 0.0; END_IF;
END_REGION

REGION Network 67: Reset TT3301_BonChua1_HMI về 0.0 khi ở chế độ chạy thật
   RUNG wire#powerrail
      I_Contact( "HMI_Sim_Mode" )
      { S7_GenerateENO := "TRUE" } Move(in := 0.0, out1 => "TT3301_BonChua1_HMI")
   END_RUNG
   // the same network as SCL:
   IF NOT "HMI_Sim_Mode" THEN "TT3301_BonChua1_HMI" := 0.0; END_IF;
END_REGION

REGION Network 68: Reset TT3303_TraoDoiNhiet_HMI về 0.0 khi ở chế độ chạy thật
   RUNG wire#powerrail
      I_Contact( "HMI_Sim_Mode" )
      { S7_GenerateENO := "TRUE" } Move(in := 0.0, out1 => "TT3303_TraoDoiNhiet_HMI")
   END_RUNG
   // the same network as SCL:
   IF NOT "HMI_Sim_Mode" THEN "TT3303_TraoDoiNhiet_HMI" := 0.0; END_IF;
END_REGION

REGION Network 69: Reset LT3307_BonChua2_HMI về 0.0 khi ở chế độ chạy thật
   RUNG wire#powerrail
      I_Contact( "HMI_Sim_Mode" )
      { S7_GenerateENO := "TRUE" } Move(in := 0.0, out1 => "LT3307_BonChua2_HMI")
   END_RUNG
   // the same network as SCL:
   IF NOT "HMI_Sim_Mode" THEN "LT3307_BonChua2_HMI" := 0.0; END_IF;
END_REGION

REGION Network 70: Reset TT3306_BonChua2_HMI về 0.0 khi ở chế độ chạy thật
   RUNG wire#powerrail
      I_Contact( "HMI_Sim_Mode" )
      { S7_GenerateENO := "TRUE" } Move(in := 0.0, out1 => "TT3306_BonChua2_HMI")
   END_RUNG
   // the same network as SCL:
   IF NOT "HMI_Sim_Mode" THEN "TT3306_BonChua2_HMI" := 0.0; END_IF;
END_REGION

REGION Network 71: Reset PI3308_Truoc_Filter_HMI về 0.0 khi ở chế độ chạy thật
   RUNG wire#powerrail
      I_Contact( "HMI_Sim_Mode" )
      { S7_GenerateENO := "TRUE" } Move(in := 0.0, out1 => "PI3308_Truoc_Filter_HMI")
   END_RUNG
   // the same network as SCL:
   IF NOT "HMI_Sim_Mode" THEN "PI3308_Truoc_Filter_HMI" := 0.0; END_IF;
END_REGION

REGION Network 72: Reset FT3309_Xa_Thanh_Pham_HMI về 0.0 khi ở chế độ chạy thật
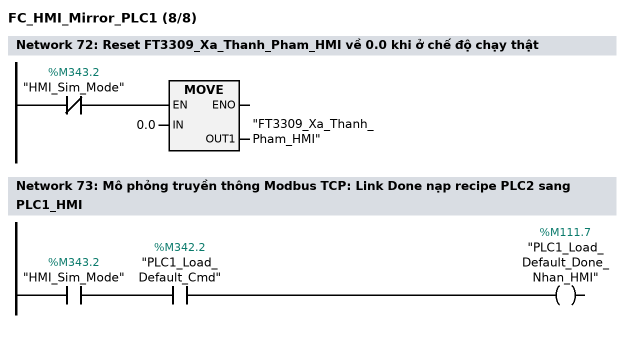
   RUNG wire#powerrail
      I_Contact( "HMI_Sim_Mode" )
      { S7_GenerateENO := "TRUE" } Move(in := 0.0, out1 => "FT3309_Xa_Thanh_Pham_HMI")
   END_RUNG
   // the same network as SCL:
   IF NOT "HMI_Sim_Mode" THEN "FT3309_Xa_Thanh_Pham_HMI" := 0.0; END_IF;
END_REGION

REGION Network 73: Mô phỏng truyền thông Modbus TCP: Link Done nạp recipe PLC2 sang PLC1_HMI
   RUNG wire#powerrail
      Contact( "HMI_Sim_Mode" )
      Contact( "PLC1_Load_Default_Cmd" )
      Coil( "PLC1_Load_Default_Done_Nhan_HMI" )
   END_RUNG
   // the same network as SCL:
   "PLC1_Load_Default_Done_Nhan_HMI" := "HMI_Sim_Mode" AND "PLC1_Load_Default_Cmd";
END_REGION
END_FUNCTION

ORGANIZATION_BLOCK "OB30_PID_PLC1_Bon2"   // OB30, LAD, CyclicInterrupt
{ S7_Optimized_Access := 'TRUE' }
VERSION : 0.1
// stored: AutoNumber true, IsIECCheckEnabled false, SetENOAutomatically false
   VAR_INPUT
      Initial_Call : Bool;   // Initial call of this OB
      Event_Count : Int;   // Events discarded
   END_VAR
BEGIN

REGION Network 1: Initialize PID Bon 2 Kp parameter
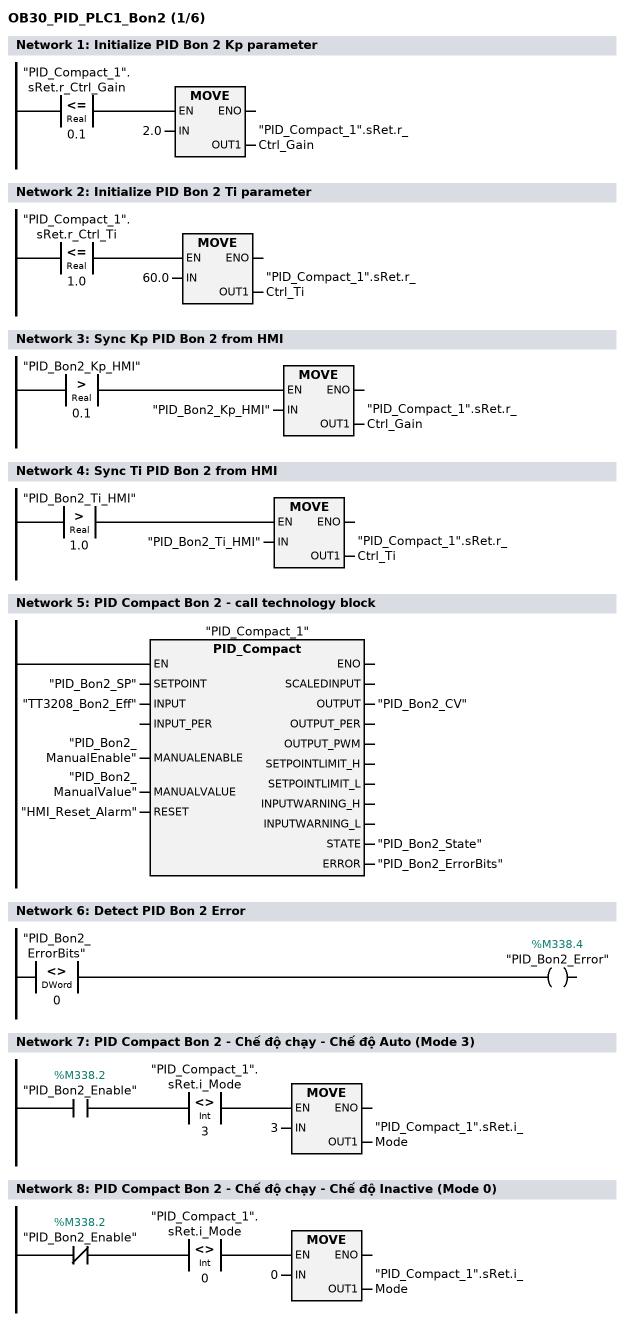
   RUNG wire#powerrail
      { S7_Templates := "SrcType := Real" } LE_Contact(in1 := "PID_Compact_1".sRet.r_Ctrl_Gain, in2 := 0.1)
      { S7_GenerateENO := "TRUE" } Move(in := 2.0, out1 => "PID_Compact_1".sRet.r_Ctrl_Gain)
   END_RUNG
   // the same network as SCL:
   IF "PID_Compact_1".sRet.r_Ctrl_Gain <= 0.1 THEN "PID_Compact_1".sRet.r_Ctrl_Gain := 2.0; END_IF;
END_REGION

REGION Network 2: Initialize PID Bon 2 Ti parameter
   RUNG wire#powerrail
      { S7_Templates := "SrcType := Real" } LE_Contact(in1 := "PID_Compact_1".sRet.r_Ctrl_Ti, in2 := 1.0)
      { S7_GenerateENO := "TRUE" } Move(in := 60.0, out1 => "PID_Compact_1".sRet.r_Ctrl_Ti)
   END_RUNG
   // the same network as SCL:
   IF "PID_Compact_1".sRet.r_Ctrl_Ti <= 1.0 THEN "PID_Compact_1".sRet.r_Ctrl_Ti := 60.0; END_IF;
END_REGION

REGION Network 3: Sync Kp PID Bon 2 from HMI
   RUNG wire#powerrail
      { S7_Templates := "SrcType := Real" } GT_Contact(in1 := "PID_Bon2_Kp_HMI", in2 := 0.1)
      { S7_GenerateENO := "TRUE" } Move(in := "PID_Bon2_Kp_HMI", out1 => "PID_Compact_1".sRet.r_Ctrl_Gain)
   END_RUNG
   // the same network as SCL:
   IF "PID_Bon2_Kp_HMI" > 0.1 THEN "PID_Compact_1".sRet.r_Ctrl_Gain := "PID_Bon2_Kp_HMI"; END_IF;
END_REGION

REGION Network 4: Sync Ti PID Bon 2 from HMI
   RUNG wire#powerrail
      { S7_Templates := "SrcType := Real" } GT_Contact(in1 := "PID_Bon2_Ti_HMI", in2 := 1.0)
      { S7_GenerateENO := "TRUE" } Move(in := "PID_Bon2_Ti_HMI", out1 => "PID_Compact_1".sRet.r_Ctrl_Ti)
   END_RUNG
   // the same network as SCL:
   IF "PID_Bon2_Ti_HMI" > 1.0 THEN "PID_Compact_1".sRet.r_Ctrl_Ti := "PID_Bon2_Ti_HMI"; END_IF;
END_REGION

REGION Network 5: PID Compact Bon 2 - call technology block
   RUNG wire#powerrail
      "PID_Compact_1".PID_Compact(Setpoint := "PID_Bon2_SP", Input := "TT3208_Bon2_Eff", Input_PER :=, ManualEnable := "PID_Bon2_ManualEnable", ManualValue := "PID_Bon2_ManualValue", Reset := "HMI_Reset_Alarm", ScaledInput =>, Output => "PID_Bon2_CV", Output_PER =>, Output_PWM =>, SetpointLimit_H =>, SetpointLimit_L =>, InputWarning_H =>, InputWarning_L =>, State => "PID_Bon2_State", Error => "PID_Bon2_ErrorBits")
   END_RUNG
   // the same network as SCL:
   "PID_Compact_1"(Setpoint := "PID_Bon2_SP",   // PID_Compact
                   Input := "TT3208_Bon2_Eff",
                   ManualEnable := "PID_Bon2_ManualEnable",
                   ManualValue := "PID_Bon2_ManualValue",
                   Reset := "HMI_Reset_Alarm",
                   Output => "PID_Bon2_CV",
                   State => "PID_Bon2_State",
                   Error => "PID_Bon2_ErrorBits");
END_REGION

REGION Network 6: Detect PID Bon 2 Error
   RUNG wire#powerrail
      { S7_Templates := "SrcType := DWord" } NE_Contact(in1 := "PID_Bon2_ErrorBits", in2 := 0)
      Coil( "PID_Bon2_Error" )
   END_RUNG
   // the same network as SCL:
   "PID_Bon2_Error" := "PID_Bon2_ErrorBits" <> 0;
END_REGION

REGION Network 7: PID Compact Bon 2 - Chế độ chạy - Chế độ Auto (Mode 3)
   RUNG wire#powerrail
      Contact( "PID_Bon2_Enable" )
      { S7_Templates := "SrcType := Int" } NE_Contact(in1 := "PID_Compact_1".sRet.i_Mode, in2 := 3)
      { S7_GenerateENO := "TRUE" } Move(in := 3, out1 => "PID_Compact_1".sRet.i_Mode)
   END_RUNG
   // the same network as SCL:
   IF "PID_Bon2_Enable" AND ("PID_Compact_1".sRet.i_Mode <> 3) THEN "PID_Compact_1".sRet.i_Mode := 3; END_IF;
END_REGION

REGION Network 8: PID Compact Bon 2 - Chế độ chạy - Chế độ Inactive (Mode 0)
   RUNG wire#powerrail
      I_Contact( "PID_Bon2_Enable" )
      { S7_Templates := "SrcType := Int" } NE_Contact(in1 := "PID_Compact_1".sRet.i_Mode, in2 := 0)
      { S7_GenerateENO := "TRUE" } Move(in := 0, out1 => "PID_Compact_1".sRet.i_Mode)
   END_RUNG
   // the same network as SCL:
   IF NOT "PID_Bon2_Enable" AND ("PID_Compact_1".sRet.i_Mode <> 0) THEN
       "PID_Compact_1".sRet.i_Mode := 0;
   END_IF;
END_REGION

REGION Network 9: Move PID Bon 2 CV to Steam Valve
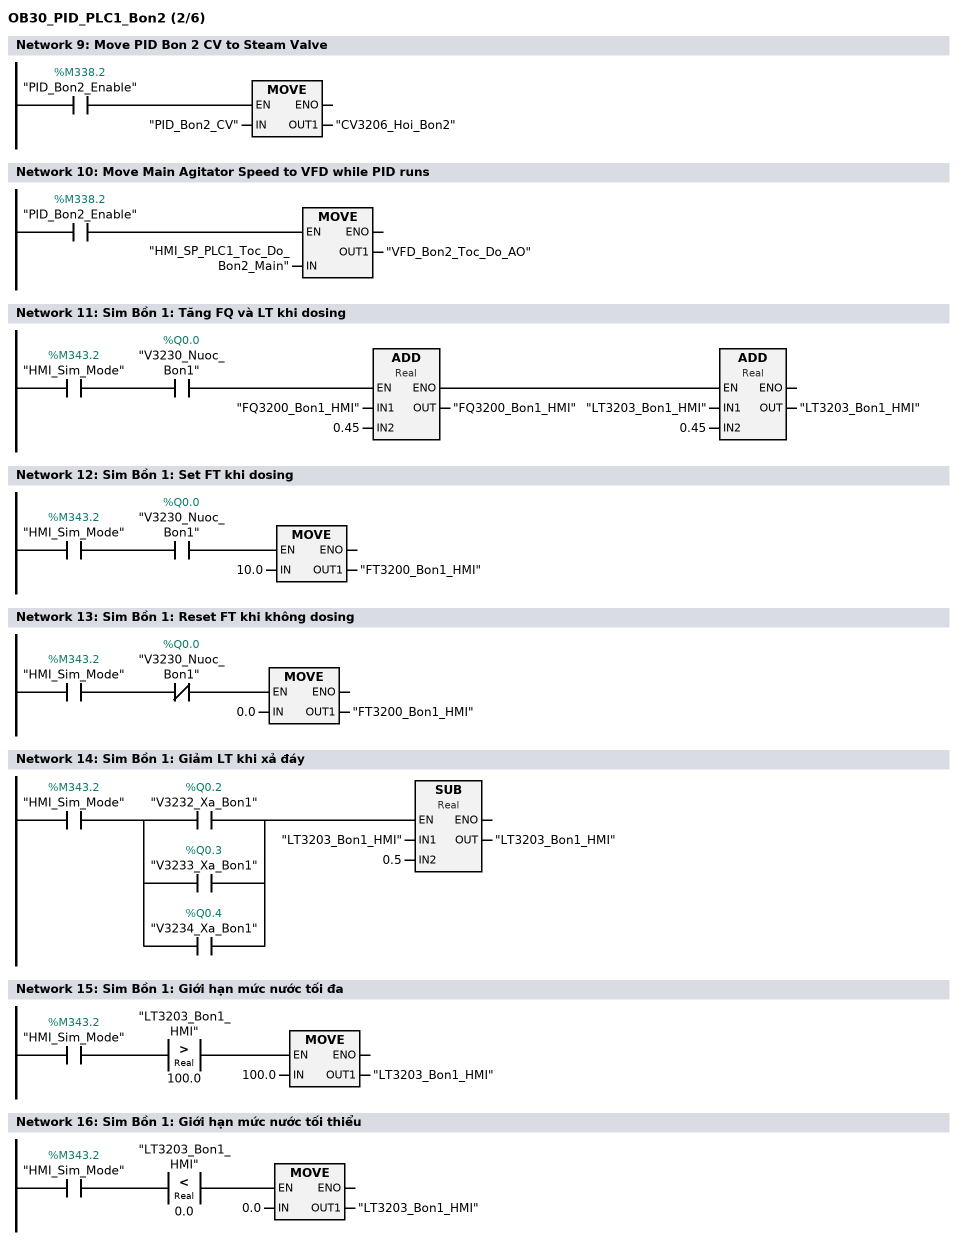
   RUNG wire#powerrail
      Contact( "PID_Bon2_Enable" )
      { S7_GenerateENO := "TRUE" } Move(in := "PID_Bon2_CV", out1 => "CV3206_Hoi_Bon2")
   END_RUNG
   // the same network as SCL:
   IF "PID_Bon2_Enable" THEN "CV3206_Hoi_Bon2" := "PID_Bon2_CV"; END_IF;
END_REGION

REGION Network 10: Move Main Agitator Speed to VFD while PID runs
   RUNG wire#powerrail
      Contact( "PID_Bon2_Enable" )
      { S7_GenerateENO := "TRUE" } Move(in := "HMI_SP_PLC1_Toc_Do_Bon2_Main", out1 => "VFD_Bon2_Toc_Do_AO")
   END_RUNG
   // the same network as SCL:
   IF "PID_Bon2_Enable" THEN "VFD_Bon2_Toc_Do_AO" := "HMI_SP_PLC1_Toc_Do_Bon2_Main"; END_IF;
END_REGION

REGION Network 11: Sim Bồn 1: Tăng FQ và LT khi dosing
   RUNG wire#powerrail
      Contact( "HMI_Sim_Mode" )
      Contact( "V3230_Nuoc_Bon1" )
      { S7_Templates := "SrcType := Real"; S7_GenerateENO := "TRUE" } Add(in1 := "FQ3200_Bon1_HMI", in2 := 0.45, out => "FQ3200_Bon1_HMI")
      { S7_Templates := "SrcType := Real"; S7_GenerateENO := "TRUE" } Add(in1 := "LT3203_Bon1_HMI", in2 := 0.45, out => "LT3203_Bon1_HMI")
   END_RUNG
   // the same network as SCL:
   // ENO of a box is taken as its EN; it also drops when the box reports an error
   IF "HMI_Sim_Mode" AND "V3230_Nuoc_Bon1" THEN
       "FQ3200_Bon1_HMI" := "FQ3200_Bon1_HMI" + 0.45;
       "LT3203_Bon1_HMI" := "LT3203_Bon1_HMI" + 0.45;
   END_IF;
END_REGION

REGION Network 12: Sim Bồn 1: Set FT khi dosing
   RUNG wire#powerrail
      Contact( "HMI_Sim_Mode" )
      Contact( "V3230_Nuoc_Bon1" )
      { S7_GenerateENO := "TRUE" } Move(in := 10.0, out1 => "FT3200_Bon1_HMI")
   END_RUNG
   // the same network as SCL:
   IF "HMI_Sim_Mode" AND "V3230_Nuoc_Bon1" THEN "FT3200_Bon1_HMI" := 10.0; END_IF;
END_REGION

REGION Network 13: Sim Bồn 1: Reset FT khi không dosing
   RUNG wire#powerrail
      Contact( "HMI_Sim_Mode" )
      I_Contact( "V3230_Nuoc_Bon1" )
      { S7_GenerateENO := "TRUE" } Move(in := 0.0, out1 => "FT3200_Bon1_HMI")
   END_RUNG
   // the same network as SCL:
   IF "HMI_Sim_Mode" AND NOT "V3230_Nuoc_Bon1" THEN "FT3200_Bon1_HMI" := 0.0; END_IF;
END_REGION

REGION Network 14: Sim Bồn 1: Giảm LT khi xả đáy
   RUNG wire#powerrail
      Contact( "HMI_Sim_Mode" )
      wire#w1
      Contact( "V3232_Xa_Bon1" )
      wire#w2
      { S7_Templates := "SrcType := Real"; S7_GenerateENO := "TRUE" } Sub(in1 := "LT3203_Bon1_HMI", in2 := 0.5, out => "LT3203_Bon1_HMI")
   END_RUNG
   RUNG wire#w1
      Contact( "V3233_Xa_Bon1" )
   END_RUNG wire#w2
   RUNG wire#w1
      Contact( "V3234_Xa_Bon1" )
   END_RUNG wire#w2
   // the same network as SCL:
   IF "HMI_Sim_Mode" AND ("V3232_Xa_Bon1" OR "V3233_Xa_Bon1" OR "V3234_Xa_Bon1") THEN
       "LT3203_Bon1_HMI" := "LT3203_Bon1_HMI" - 0.5;
   END_IF;
END_REGION

REGION Network 15: Sim Bồn 1: Giới hạn mức nước tối đa
   RUNG wire#powerrail
      Contact( "HMI_Sim_Mode" )
      { S7_Templates := "SrcType := Real" } GT_Contact(in1 := "LT3203_Bon1_HMI", in2 := 100.0)
      { S7_GenerateENO := "TRUE" } Move(in := 100.0, out1 => "LT3203_Bon1_HMI")
   END_RUNG
   // the same network as SCL:
   IF "HMI_Sim_Mode" AND ("LT3203_Bon1_HMI" > 100.0) THEN "LT3203_Bon1_HMI" := 100.0; END_IF;
END_REGION

REGION Network 16: Sim Bồn 1: Giới hạn mức nước tối thiểu
   RUNG wire#powerrail
      Contact( "HMI_Sim_Mode" )
      { S7_Templates := "SrcType := Real" } LT_Contact(in1 := "LT3203_Bon1_HMI", in2 := 0.0)
      { S7_GenerateENO := "TRUE" } Move(in := 0.0, out1 => "LT3203_Bon1_HMI")
   END_RUNG
   // the same network as SCL:
   IF "HMI_Sim_Mode" AND ("LT3203_Bon1_HMI" < 0.0) THEN "LT3203_Bon1_HMI" := 0.0; END_IF;
END_REGION

REGION Network 17: Sim Bồn 2: Tăng FQ và LT khi dosing
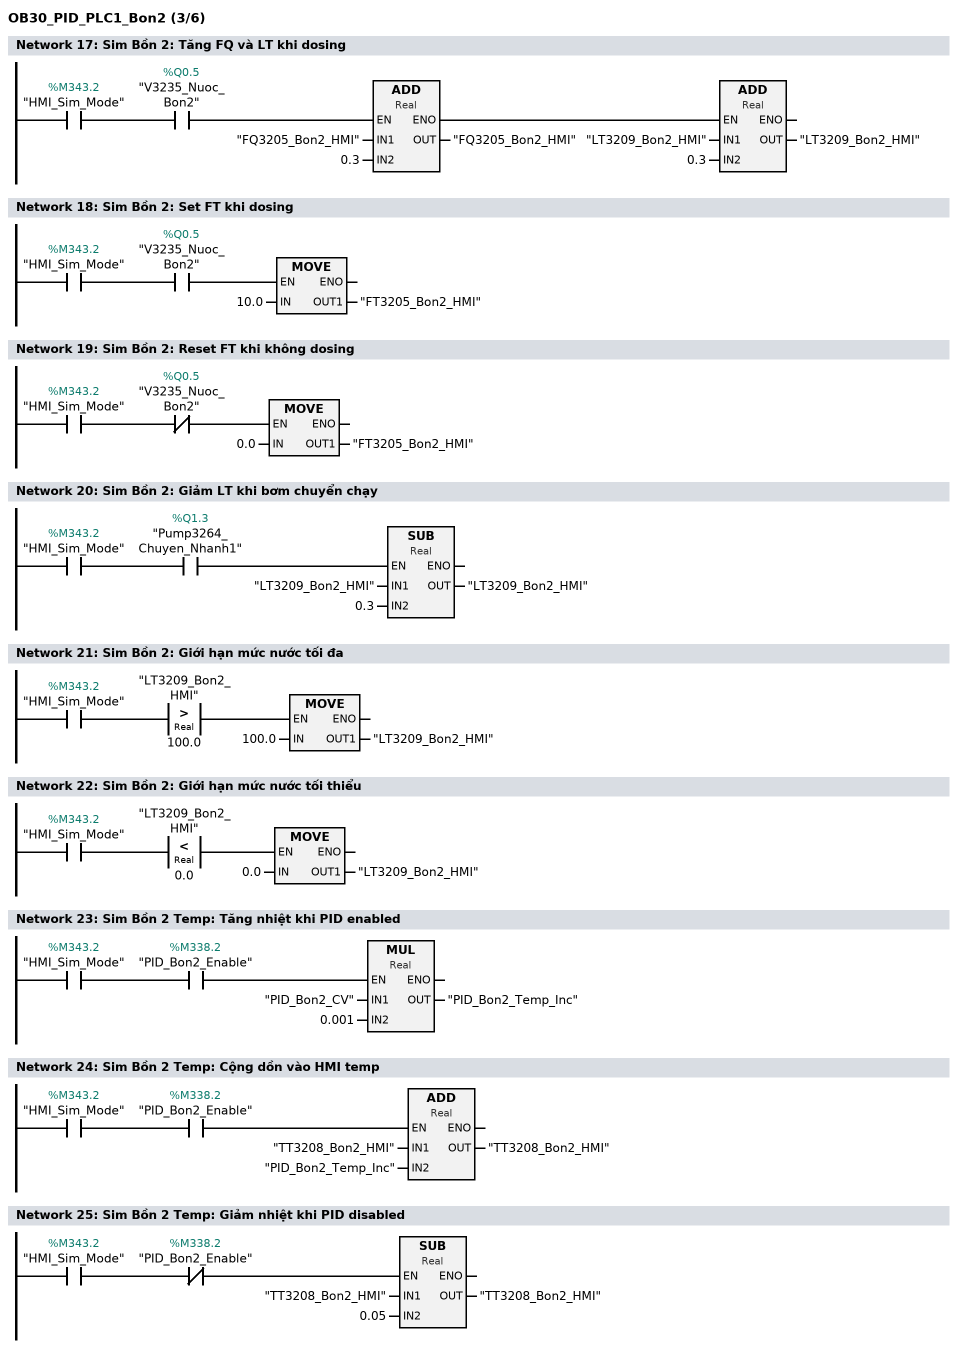
   RUNG wire#powerrail
      Contact( "HMI_Sim_Mode" )
      Contact( "V3235_Nuoc_Bon2" )
      { S7_Templates := "SrcType := Real"; S7_GenerateENO := "TRUE" } Add(in1 := "FQ3205_Bon2_HMI", in2 := 0.3, out => "FQ3205_Bon2_HMI")
      { S7_Templates := "SrcType := Real"; S7_GenerateENO := "TRUE" } Add(in1 := "LT3209_Bon2_HMI", in2 := 0.3, out => "LT3209_Bon2_HMI")
   END_RUNG
   // the same network as SCL:
   // ENO of a box is taken as its EN; it also drops when the box reports an error
   IF "HMI_Sim_Mode" AND "V3235_Nuoc_Bon2" THEN
       "FQ3205_Bon2_HMI" := "FQ3205_Bon2_HMI" + 0.3;
       "LT3209_Bon2_HMI" := "LT3209_Bon2_HMI" + 0.3;
   END_IF;
END_REGION

REGION Network 18: Sim Bồn 2: Set FT khi dosing
   RUNG wire#powerrail
      Contact( "HMI_Sim_Mode" )
      Contact( "V3235_Nuoc_Bon2" )
      { S7_GenerateENO := "TRUE" } Move(in := 10.0, out1 => "FT3205_Bon2_HMI")
   END_RUNG
   // the same network as SCL:
   IF "HMI_Sim_Mode" AND "V3235_Nuoc_Bon2" THEN "FT3205_Bon2_HMI" := 10.0; END_IF;
END_REGION

REGION Network 19: Sim Bồn 2: Reset FT khi không dosing
   RUNG wire#powerrail
      Contact( "HMI_Sim_Mode" )
      I_Contact( "V3235_Nuoc_Bon2" )
      { S7_GenerateENO := "TRUE" } Move(in := 0.0, out1 => "FT3205_Bon2_HMI")
   END_RUNG
   // the same network as SCL:
   IF "HMI_Sim_Mode" AND NOT "V3235_Nuoc_Bon2" THEN "FT3205_Bon2_HMI" := 0.0; END_IF;
END_REGION

REGION Network 20: Sim Bồn 2: Giảm LT khi bơm chuyển chạy
   RUNG wire#powerrail
      Contact( "HMI_Sim_Mode" )
      Contact( "Pump3264_Chuyen_Nhanh1" )
      { S7_Templates := "SrcType := Real"; S7_GenerateENO := "TRUE" } Sub(in1 := "LT3209_Bon2_HMI", in2 := 0.3, out => "LT3209_Bon2_HMI")
   END_RUNG
   // the same network as SCL:
   IF "HMI_Sim_Mode" AND "Pump3264_Chuyen_Nhanh1" THEN "LT3209_Bon2_HMI" := "LT3209_Bon2_HMI" - 0.3; END_IF;
END_REGION

REGION Network 21: Sim Bồn 2: Giới hạn mức nước tối đa
   RUNG wire#powerrail
      Contact( "HMI_Sim_Mode" )
      { S7_Templates := "SrcType := Real" } GT_Contact(in1 := "LT3209_Bon2_HMI", in2 := 100.0)
      { S7_GenerateENO := "TRUE" } Move(in := 100.0, out1 => "LT3209_Bon2_HMI")
   END_RUNG
   // the same network as SCL:
   IF "HMI_Sim_Mode" AND ("LT3209_Bon2_HMI" > 100.0) THEN "LT3209_Bon2_HMI" := 100.0; END_IF;
END_REGION

REGION Network 22: Sim Bồn 2: Giới hạn mức nước tối thiểu
   RUNG wire#powerrail
      Contact( "HMI_Sim_Mode" )
      { S7_Templates := "SrcType := Real" } LT_Contact(in1 := "LT3209_Bon2_HMI", in2 := 0.0)
      { S7_GenerateENO := "TRUE" } Move(in := 0.0, out1 => "LT3209_Bon2_HMI")
   END_RUNG
   // the same network as SCL:
   IF "HMI_Sim_Mode" AND ("LT3209_Bon2_HMI" < 0.0) THEN "LT3209_Bon2_HMI" := 0.0; END_IF;
END_REGION

REGION Network 23: Sim Bồn 2 Temp: Tăng nhiệt khi PID enabled
   RUNG wire#powerrail
      Contact( "HMI_Sim_Mode" )
      Contact( "PID_Bon2_Enable" )
      { S7_Templates := "SrcType := Real"; S7_GenerateENO := "TRUE" } Mul(in1 := "PID_Bon2_CV", in2 := 0.001, out => "PID_Bon2_Temp_Inc")
   END_RUNG
   // the same network as SCL:
   IF "HMI_Sim_Mode" AND "PID_Bon2_Enable" THEN "PID_Bon2_Temp_Inc" := "PID_Bon2_CV" * 0.001; END_IF;
END_REGION

REGION Network 24: Sim Bồn 2 Temp: Cộng dồn vào HMI temp
   RUNG wire#powerrail
      Contact( "HMI_Sim_Mode" )
      Contact( "PID_Bon2_Enable" )
      { S7_Templates := "SrcType := Real"; S7_GenerateENO := "TRUE" } Add(in1 := "TT3208_Bon2_HMI", in2 := "PID_Bon2_Temp_Inc", out => "TT3208_Bon2_HMI")
   END_RUNG
   // the same network as SCL:
   IF "HMI_Sim_Mode" AND "PID_Bon2_Enable" THEN
       "TT3208_Bon2_HMI" := "TT3208_Bon2_HMI" + "PID_Bon2_Temp_Inc";
   END_IF;
END_REGION

REGION Network 25: Sim Bồn 2 Temp: Giảm nhiệt khi PID disabled
   RUNG wire#powerrail
      Contact( "HMI_Sim_Mode" )
      I_Contact( "PID_Bon2_Enable" )
      { S7_Templates := "SrcType := Real"; S7_GenerateENO := "TRUE" } Sub(in1 := "TT3208_Bon2_HMI", in2 := 0.05, out => "TT3208_Bon2_HMI")
   END_RUNG
   // the same network as SCL:
   IF "HMI_Sim_Mode" AND NOT "PID_Bon2_Enable" THEN "TT3208_Bon2_HMI" := "TT3208_Bon2_HMI" - 0.05; END_IF;
END_REGION

REGION Network 26: Sim Bồn 2 Temp: Giới hạn nhiệt độ tối đa 100
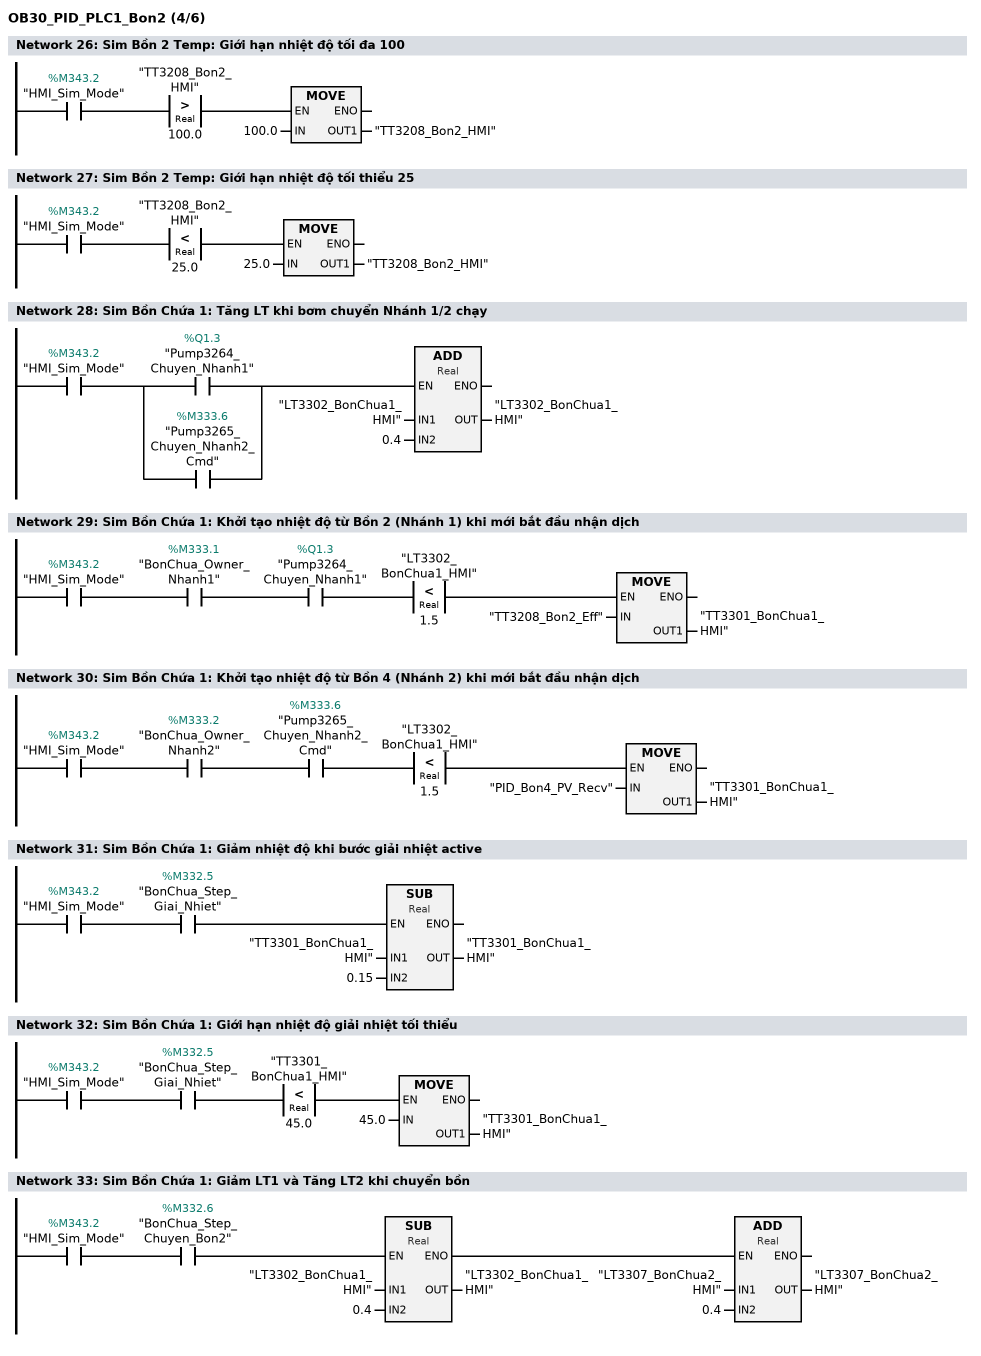
   RUNG wire#powerrail
      Contact( "HMI_Sim_Mode" )
      { S7_Templates := "SrcType := Real" } GT_Contact(in1 := "TT3208_Bon2_HMI", in2 := 100.0)
      { S7_GenerateENO := "TRUE" } Move(in := 100.0, out1 => "TT3208_Bon2_HMI")
   END_RUNG
   // the same network as SCL:
   IF "HMI_Sim_Mode" AND ("TT3208_Bon2_HMI" > 100.0) THEN "TT3208_Bon2_HMI" := 100.0; END_IF;
END_REGION

REGION Network 27: Sim Bồn 2 Temp: Giới hạn nhiệt độ tối thiểu 25
   RUNG wire#powerrail
      Contact( "HMI_Sim_Mode" )
      { S7_Templates := "SrcType := Real" } LT_Contact(in1 := "TT3208_Bon2_HMI", in2 := 25.0)
      { S7_GenerateENO := "TRUE" } Move(in := 25.0, out1 => "TT3208_Bon2_HMI")
   END_RUNG
   // the same network as SCL:
   IF "HMI_Sim_Mode" AND ("TT3208_Bon2_HMI" < 25.0) THEN "TT3208_Bon2_HMI" := 25.0; END_IF;
END_REGION

REGION Network 28: Sim Bồn Chứa 1: Tăng LT khi bơm chuyển Nhánh 1/2 chạy
   RUNG wire#powerrail
      Contact( "HMI_Sim_Mode" )
      wire#w1
      Contact( "Pump3264_Chuyen_Nhanh1" )
      wire#w2
      { S7_Templates := "SrcType := Real"; S7_GenerateENO := "TRUE" } Add(in1 := "LT3302_BonChua1_HMI", in2 := 0.4, out => "LT3302_BonChua1_HMI")
   END_RUNG
   RUNG wire#w1
      Contact( "Pump3265_Chuyen_Nhanh2_Cmd" )
   END_RUNG wire#w2
   // the same network as SCL:
   IF "HMI_Sim_Mode" AND ("Pump3264_Chuyen_Nhanh1" OR "Pump3265_Chuyen_Nhanh2_Cmd") THEN
       "LT3302_BonChua1_HMI" := "LT3302_BonChua1_HMI" + 0.4;
   END_IF;
END_REGION

REGION Network 29: Sim Bồn Chứa 1: Khởi tạo nhiệt độ từ Bồn 2 (Nhánh 1) khi mới bắt đầu nhận dịch
   RUNG wire#powerrail
      Contact( "HMI_Sim_Mode" )
      Contact( "BonChua_Owner_Nhanh1" )
      Contact( "Pump3264_Chuyen_Nhanh1" )
      { S7_Templates := "SrcType := Real" } LT_Contact(in1 := "LT3302_BonChua1_HMI", in2 := 1.5)
      { S7_GenerateENO := "TRUE" } Move(in := "TT3208_Bon2_Eff", out1 => "TT3301_BonChua1_HMI")
   END_RUNG
   // the same network as SCL:
   IF "HMI_Sim_Mode" AND "BonChua_Owner_Nhanh1" AND "Pump3264_Chuyen_Nhanh1" AND ("LT3302_BonChua1_HMI" < 1.5) THEN
       "TT3301_BonChua1_HMI" := "TT3208_Bon2_Eff";
   END_IF;
END_REGION

REGION Network 30: Sim Bồn Chứa 1: Khởi tạo nhiệt độ từ Bồn 4 (Nhánh 2) khi mới bắt đầu nhận dịch
   RUNG wire#powerrail
      Contact( "HMI_Sim_Mode" )
      Contact( "BonChua_Owner_Nhanh2" )
      Contact( "Pump3265_Chuyen_Nhanh2_Cmd" )
      { S7_Templates := "SrcType := Real" } LT_Contact(in1 := "LT3302_BonChua1_HMI", in2 := 1.5)
      { S7_GenerateENO := "TRUE" } Move(in := "PID_Bon4_PV_Recv", out1 => "TT3301_BonChua1_HMI")
   END_RUNG
   // the same network as SCL:
   IF "HMI_Sim_Mode" AND "BonChua_Owner_Nhanh2" AND "Pump3265_Chuyen_Nhanh2_Cmd" AND ("LT3302_BonChua1_HMI" < 1.5) THEN
       "TT3301_BonChua1_HMI" := "PID_Bon4_PV_Recv";
   END_IF;
END_REGION

REGION Network 31: Sim Bồn Chứa 1: Giảm nhiệt độ khi bước giải nhiệt active
   RUNG wire#powerrail
      Contact( "HMI_Sim_Mode" )
      Contact( "BonChua_Step_Giai_Nhiet" )
      { S7_Templates := "SrcType := Real"; S7_GenerateENO := "TRUE" } Sub(in1 := "TT3301_BonChua1_HMI", in2 := 0.15, out => "TT3301_BonChua1_HMI")
   END_RUNG
   // the same network as SCL:
   IF "HMI_Sim_Mode" AND "BonChua_Step_Giai_Nhiet" THEN
       "TT3301_BonChua1_HMI" := "TT3301_BonChua1_HMI" - 0.15;
   END_IF;
END_REGION

REGION Network 32: Sim Bồn Chứa 1: Giới hạn nhiệt độ giải nhiệt tối thiểu
   RUNG wire#powerrail
      Contact( "HMI_Sim_Mode" )
      Contact( "BonChua_Step_Giai_Nhiet" )
      { S7_Templates := "SrcType := Real" } LT_Contact(in1 := "TT3301_BonChua1_HMI", in2 := 45.0)
      { S7_GenerateENO := "TRUE" } Move(in := 45.0, out1 => "TT3301_BonChua1_HMI")
   END_RUNG
   // the same network as SCL:
   IF "HMI_Sim_Mode" AND "BonChua_Step_Giai_Nhiet" AND ("TT3301_BonChua1_HMI" < 45.0) THEN
       "TT3301_BonChua1_HMI" := 45.0;
   END_IF;
END_REGION

REGION Network 33: Sim Bồn Chứa 1: Giảm LT1 và Tăng LT2 khi chuyển bồn
   RUNG wire#powerrail
      Contact( "HMI_Sim_Mode" )
      Contact( "BonChua_Step_Chuyen_Bon2" )
      { S7_Templates := "SrcType := Real"; S7_GenerateENO := "TRUE" } Sub(in1 := "LT3302_BonChua1_HMI", in2 := 0.4, out => "LT3302_BonChua1_HMI")
      { S7_Templates := "SrcType := Real"; S7_GenerateENO := "TRUE" } Add(in1 := "LT3307_BonChua2_HMI", in2 := 0.4, out => "LT3307_BonChua2_HMI")
   END_RUNG
   // the same network as SCL:
   // ENO of a box is taken as its EN; it also drops when the box reports an error
   IF "HMI_Sim_Mode" AND "BonChua_Step_Chuyen_Bon2" THEN
       "LT3302_BonChua1_HMI" := "LT3302_BonChua1_HMI" - 0.4;
       "LT3307_BonChua2_HMI" := "LT3307_BonChua2_HMI" + 0.4;
   END_IF;
END_REGION

REGION Network 34: Sim Bồn Chứa 1: Tự động kết thúc bước chuyển bồn
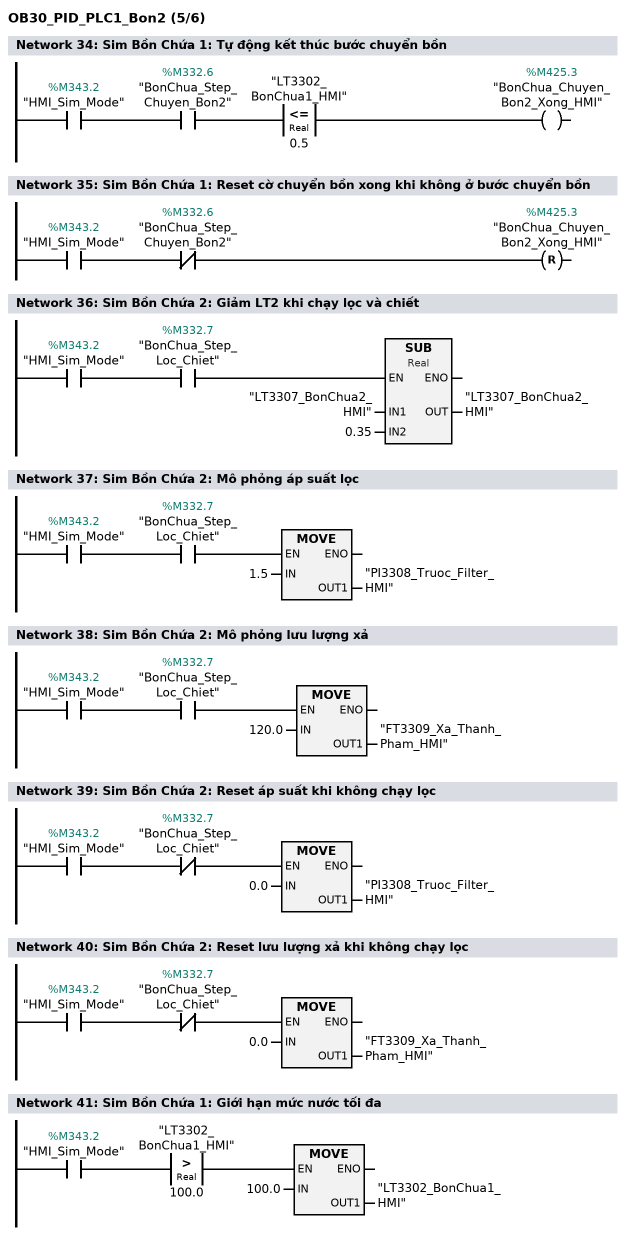
   RUNG wire#powerrail
      Contact( "HMI_Sim_Mode" )
      Contact( "BonChua_Step_Chuyen_Bon2" )
      { S7_Templates := "SrcType := Real" } LE_Contact(in1 := "LT3302_BonChua1_HMI", in2 := 0.5)
      Coil( "BonChua_Chuyen_Bon2_Xong_HMI" )
   END_RUNG
   // the same network as SCL:
   "BonChua_Chuyen_Bon2_Xong_HMI" := "HMI_Sim_Mode" AND "BonChua_Step_Chuyen_Bon2" AND ("LT3302_BonChua1_HMI" <= 0.5);
END_REGION

REGION Network 35: Sim Bồn Chứa 1: Reset cờ chuyển bồn xong khi không ở bước chuyển bồn
   RUNG wire#powerrail
      Contact( "HMI_Sim_Mode" )
      I_Contact( "BonChua_Step_Chuyen_Bon2" )
      R_Coil( "BonChua_Chuyen_Bon2_Xong_HMI" )
   END_RUNG
   // the same network as SCL:
   IF "HMI_Sim_Mode" AND NOT "BonChua_Step_Chuyen_Bon2" THEN "BonChua_Chuyen_Bon2_Xong_HMI" := FALSE; END_IF;
END_REGION

REGION Network 36: Sim Bồn Chứa 2: Giảm LT2 khi chạy lọc và chiết
   RUNG wire#powerrail
      Contact( "HMI_Sim_Mode" )
      Contact( "BonChua_Step_Loc_Chiet" )
      { S7_Templates := "SrcType := Real"; S7_GenerateENO := "TRUE" } Sub(in1 := "LT3307_BonChua2_HMI", in2 := 0.35, out => "LT3307_BonChua2_HMI")
   END_RUNG
   // the same network as SCL:
   IF "HMI_Sim_Mode" AND "BonChua_Step_Loc_Chiet" THEN
       "LT3307_BonChua2_HMI" := "LT3307_BonChua2_HMI" - 0.35;
   END_IF;
END_REGION

REGION Network 37: Sim Bồn Chứa 2: Mô phỏng áp suất lọc
   RUNG wire#powerrail
      Contact( "HMI_Sim_Mode" )
      Contact( "BonChua_Step_Loc_Chiet" )
      { S7_GenerateENO := "TRUE" } Move(in := 1.5, out1 => "PI3308_Truoc_Filter_HMI")
   END_RUNG
   // the same network as SCL:
   IF "HMI_Sim_Mode" AND "BonChua_Step_Loc_Chiet" THEN "PI3308_Truoc_Filter_HMI" := 1.5; END_IF;
END_REGION

REGION Network 38: Sim Bồn Chứa 2: Mô phỏng lưu lượng xả
   RUNG wire#powerrail
      Contact( "HMI_Sim_Mode" )
      Contact( "BonChua_Step_Loc_Chiet" )
      { S7_GenerateENO := "TRUE" } Move(in := 120.0, out1 => "FT3309_Xa_Thanh_Pham_HMI")
   END_RUNG
   // the same network as SCL:
   IF "HMI_Sim_Mode" AND "BonChua_Step_Loc_Chiet" THEN "FT3309_Xa_Thanh_Pham_HMI" := 120.0; END_IF;
END_REGION

REGION Network 39: Sim Bồn Chứa 2: Reset áp suất khi không chạy lọc
   RUNG wire#powerrail
      Contact( "HMI_Sim_Mode" )
      I_Contact( "BonChua_Step_Loc_Chiet" )
      { S7_GenerateENO := "TRUE" } Move(in := 0.0, out1 => "PI3308_Truoc_Filter_HMI")
   END_RUNG
   // the same network as SCL:
   IF "HMI_Sim_Mode" AND NOT "BonChua_Step_Loc_Chiet" THEN "PI3308_Truoc_Filter_HMI" := 0.0; END_IF;
END_REGION

REGION Network 40: Sim Bồn Chứa 2: Reset lưu lượng xả khi không chạy lọc
   RUNG wire#powerrail
      Contact( "HMI_Sim_Mode" )
      I_Contact( "BonChua_Step_Loc_Chiet" )
      { S7_GenerateENO := "TRUE" } Move(in := 0.0, out1 => "FT3309_Xa_Thanh_Pham_HMI")
   END_RUNG
   // the same network as SCL:
   IF "HMI_Sim_Mode" AND NOT "BonChua_Step_Loc_Chiet" THEN "FT3309_Xa_Thanh_Pham_HMI" := 0.0; END_IF;
END_REGION

REGION Network 41: Sim Bồn Chứa 1: Giới hạn mức nước tối đa
   RUNG wire#powerrail
      Contact( "HMI_Sim_Mode" )
      { S7_Templates := "SrcType := Real" } GT_Contact(in1 := "LT3302_BonChua1_HMI", in2 := 100.0)
      { S7_GenerateENO := "TRUE" } Move(in := 100.0, out1 => "LT3302_BonChua1_HMI")
   END_RUNG
   // the same network as SCL:
   IF "HMI_Sim_Mode" AND ("LT3302_BonChua1_HMI" > 100.0) THEN "LT3302_BonChua1_HMI" := 100.0; END_IF;
END_REGION

REGION Network 42: Sim Bồn Chứa 1: Giới hạn mức nước tối thiểu
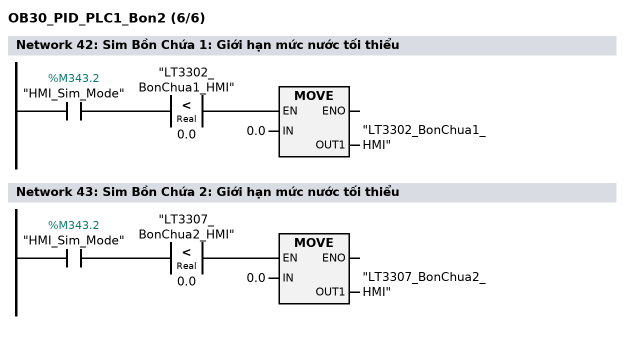
   RUNG wire#powerrail
      Contact( "HMI_Sim_Mode" )
      { S7_Templates := "SrcType := Real" } LT_Contact(in1 := "LT3302_BonChua1_HMI", in2 := 0.0)
      { S7_GenerateENO := "TRUE" } Move(in := 0.0, out1 => "LT3302_BonChua1_HMI")
   END_RUNG
   // the same network as SCL:
   IF "HMI_Sim_Mode" AND ("LT3302_BonChua1_HMI" < 0.0) THEN "LT3302_BonChua1_HMI" := 0.0; END_IF;
END_REGION

REGION Network 43: Sim Bồn Chứa 2: Giới hạn mức nước tối thiểu
   RUNG wire#powerrail
      Contact( "HMI_Sim_Mode" )
      { S7_Templates := "SrcType := Real" } LT_Contact(in1 := "LT3307_BonChua2_HMI", in2 := 0.0)
      { S7_GenerateENO := "TRUE" } Move(in := 0.0, out1 => "LT3307_BonChua2_HMI")
   END_RUNG
   // the same network as SCL:
   IF "HMI_Sim_Mode" AND ("LT3307_BonChua2_HMI" < 0.0) THEN "LT3307_BonChua2_HMI" := 0.0; END_IF;
END_REGION
END_ORGANIZATION_BLOCK

ORGANIZATION_BLOCK "OB31_PID_PLC2_Bon4"   // OB31, LAD, CyclicInterrupt
{ S7_Optimized_Access := 'TRUE' }
VERSION : 0.1
// stored: AutoNumber true, IsIECCheckEnabled false, SetENOAutomatically false
   VAR_INPUT
      Initial_Call : Bool;   // Initial call of this OB
      Event_Count : Int;   // Events discarded
   END_VAR
BEGIN

REGION Network 1: Initialize PID Bon 4 Kp parameter
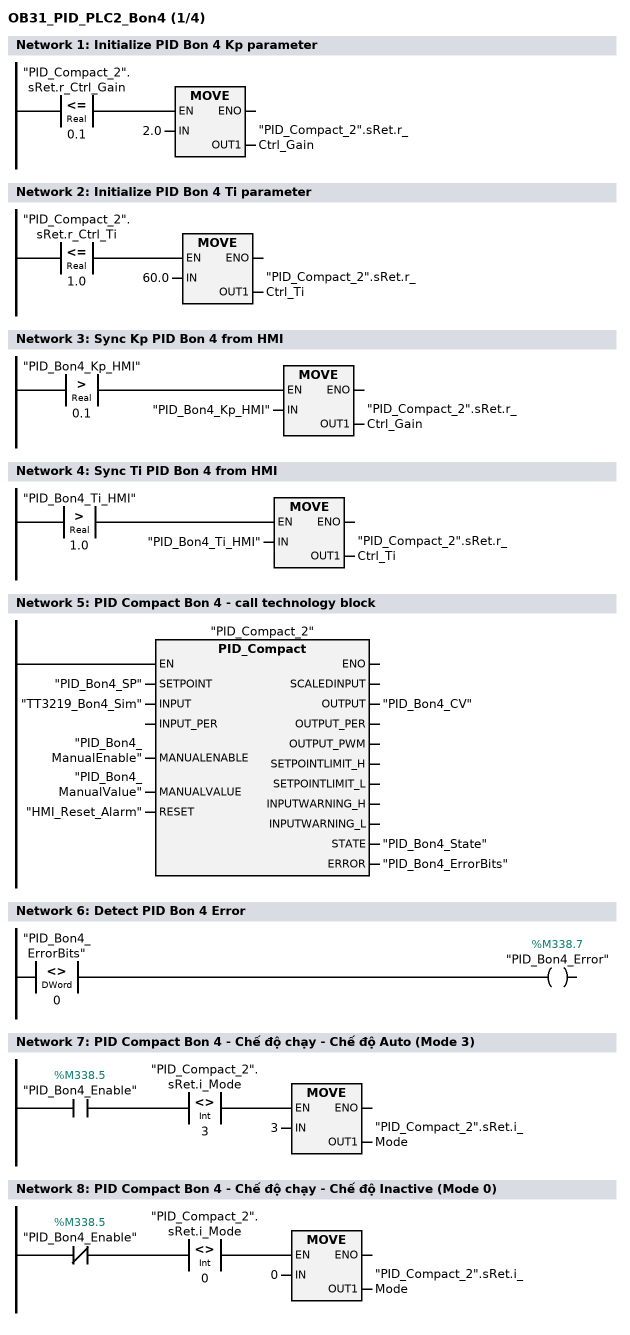
   RUNG wire#powerrail
      { S7_Templates := "SrcType := Real" } LE_Contact(in1 := "PID_Compact_2".sRet.r_Ctrl_Gain, in2 := 0.1)
      { S7_GenerateENO := "TRUE" } Move(in := 2.0, out1 => "PID_Compact_2".sRet.r_Ctrl_Gain)
   END_RUNG
   // the same network as SCL:
   IF "PID_Compact_2".sRet.r_Ctrl_Gain <= 0.1 THEN "PID_Compact_2".sRet.r_Ctrl_Gain := 2.0; END_IF;
END_REGION

REGION Network 2: Initialize PID Bon 4 Ti parameter
   RUNG wire#powerrail
      { S7_Templates := "SrcType := Real" } LE_Contact(in1 := "PID_Compact_2".sRet.r_Ctrl_Ti, in2 := 1.0)
      { S7_GenerateENO := "TRUE" } Move(in := 60.0, out1 => "PID_Compact_2".sRet.r_Ctrl_Ti)
   END_RUNG
   // the same network as SCL:
   IF "PID_Compact_2".sRet.r_Ctrl_Ti <= 1.0 THEN "PID_Compact_2".sRet.r_Ctrl_Ti := 60.0; END_IF;
END_REGION

REGION Network 3: Sync Kp PID Bon 4 from HMI
   RUNG wire#powerrail
      { S7_Templates := "SrcType := Real" } GT_Contact(in1 := "PID_Bon4_Kp_HMI", in2 := 0.1)
      { S7_GenerateENO := "TRUE" } Move(in := "PID_Bon4_Kp_HMI", out1 => "PID_Compact_2".sRet.r_Ctrl_Gain)
   END_RUNG
   // the same network as SCL:
   IF "PID_Bon4_Kp_HMI" > 0.1 THEN "PID_Compact_2".sRet.r_Ctrl_Gain := "PID_Bon4_Kp_HMI"; END_IF;
END_REGION

REGION Network 4: Sync Ti PID Bon 4 from HMI
   RUNG wire#powerrail
      { S7_Templates := "SrcType := Real" } GT_Contact(in1 := "PID_Bon4_Ti_HMI", in2 := 1.0)
      { S7_GenerateENO := "TRUE" } Move(in := "PID_Bon4_Ti_HMI", out1 => "PID_Compact_2".sRet.r_Ctrl_Ti)
   END_RUNG
   // the same network as SCL:
   IF "PID_Bon4_Ti_HMI" > 1.0 THEN "PID_Compact_2".sRet.r_Ctrl_Ti := "PID_Bon4_Ti_HMI"; END_IF;
END_REGION

REGION Network 5: PID Compact Bon 4 - call technology block
   RUNG wire#powerrail
      "PID_Compact_2".PID_Compact(Setpoint := "PID_Bon4_SP", Input := "TT3219_Bon4_Sim", Input_PER :=, ManualEnable := "PID_Bon4_ManualEnable", ManualValue := "PID_Bon4_ManualValue", Reset := "HMI_Reset_Alarm", ScaledInput =>, Output => "PID_Bon4_CV", Output_PER =>, Output_PWM =>, SetpointLimit_H =>, SetpointLimit_L =>, InputWarning_H =>, InputWarning_L =>, State => "PID_Bon4_State", Error => "PID_Bon4_ErrorBits")
   END_RUNG
   // the same network as SCL:
   "PID_Compact_2"(Setpoint := "PID_Bon4_SP",   // PID_Compact
                   Input := "TT3219_Bon4_Sim",
                   ManualEnable := "PID_Bon4_ManualEnable",
                   ManualValue := "PID_Bon4_ManualValue",
                   Reset := "HMI_Reset_Alarm",
                   Output => "PID_Bon4_CV",
                   State => "PID_Bon4_State",
                   Error => "PID_Bon4_ErrorBits");
END_REGION

REGION Network 6: Detect PID Bon 4 Error
   RUNG wire#powerrail
      { S7_Templates := "SrcType := DWord" } NE_Contact(in1 := "PID_Bon4_ErrorBits", in2 := 0)
      Coil( "PID_Bon4_Error" )
   END_RUNG
   // the same network as SCL:
   "PID_Bon4_Error" := "PID_Bon4_ErrorBits" <> 0;
END_REGION

REGION Network 7: PID Compact Bon 4 - Chế độ chạy - Chế độ Auto (Mode 3)
   RUNG wire#powerrail
      Contact( "PID_Bon4_Enable" )
      { S7_Templates := "SrcType := Int" } NE_Contact(in1 := "PID_Compact_2".sRet.i_Mode, in2 := 3)
      { S7_GenerateENO := "TRUE" } Move(in := 3, out1 => "PID_Compact_2".sRet.i_Mode)
   END_RUNG
   // the same network as SCL:
   IF "PID_Bon4_Enable" AND ("PID_Compact_2".sRet.i_Mode <> 3) THEN "PID_Compact_2".sRet.i_Mode := 3; END_IF;
END_REGION

REGION Network 8: PID Compact Bon 4 - Chế độ chạy - Chế độ Inactive (Mode 0)
   RUNG wire#powerrail
      I_Contact( "PID_Bon4_Enable" )
      { S7_Templates := "SrcType := Int" } NE_Contact(in1 := "PID_Compact_2".sRet.i_Mode, in2 := 0)
      { S7_GenerateENO := "TRUE" } Move(in := 0, out1 => "PID_Compact_2".sRet.i_Mode)
   END_RUNG
   // the same network as SCL:
   IF NOT "PID_Bon4_Enable" AND ("PID_Compact_2".sRet.i_Mode <> 0) THEN
       "PID_Compact_2".sRet.i_Mode := 0;
   END_IF;
END_REGION

REGION Network 9: Move PID Bon 4 CV to simulated heat valve
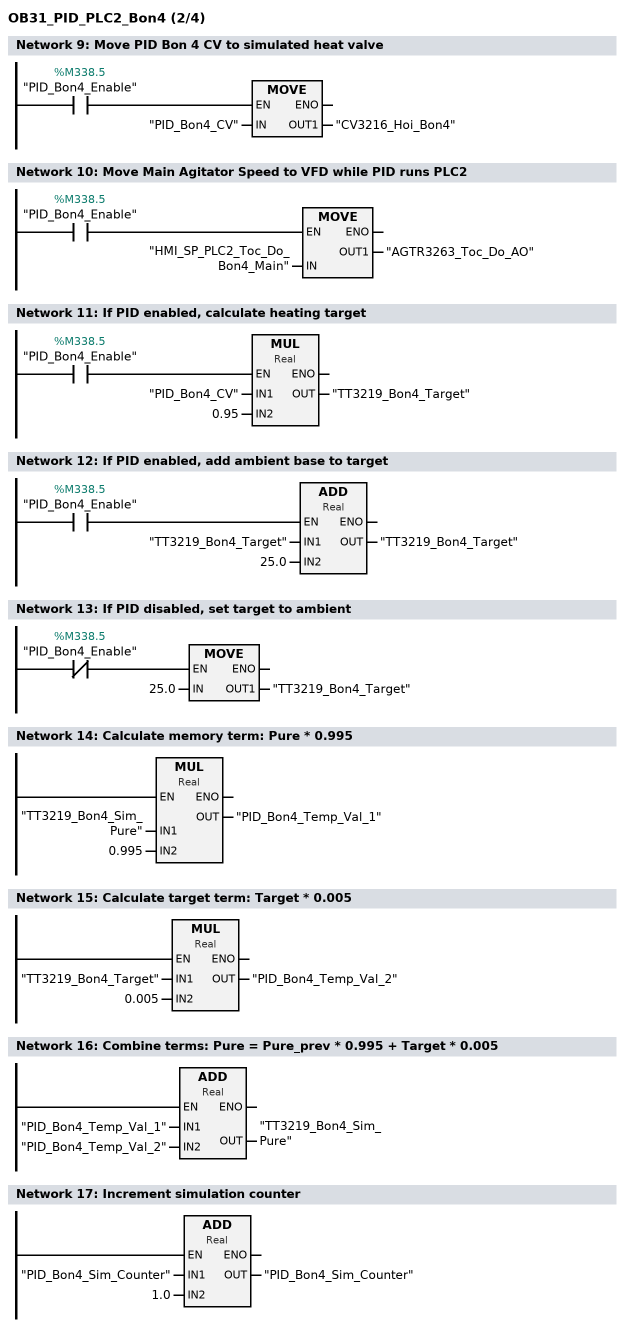
   RUNG wire#powerrail
      Contact( "PID_Bon4_Enable" )
      { S7_GenerateENO := "TRUE" } Move(in := "PID_Bon4_CV", out1 => "CV3216_Hoi_Bon4")
   END_RUNG
   // the same network as SCL:
   IF "PID_Bon4_Enable" THEN "CV3216_Hoi_Bon4" := "PID_Bon4_CV"; END_IF;
END_REGION

REGION Network 10: Move Main Agitator Speed to VFD while PID runs PLC2
   RUNG wire#powerrail
      Contact( "PID_Bon4_Enable" )
      { S7_GenerateENO := "TRUE" } Move(in := "HMI_SP_PLC2_Toc_Do_Bon4_Main", out1 => "AGTR3263_Toc_Do_AO")
   END_RUNG
   // the same network as SCL:
   IF "PID_Bon4_Enable" THEN "AGTR3263_Toc_Do_AO" := "HMI_SP_PLC2_Toc_Do_Bon4_Main"; END_IF;
END_REGION

REGION Network 11: If PID enabled, calculate heating target
   RUNG wire#powerrail
      Contact( "PID_Bon4_Enable" )
      { S7_Templates := "SrcType := Real"; S7_GenerateENO := "TRUE" } Mul(in1 := "PID_Bon4_CV", in2 := 0.95, out => "TT3219_Bon4_Target")
   END_RUNG
   // the same network as SCL:
   IF "PID_Bon4_Enable" THEN "TT3219_Bon4_Target" := "PID_Bon4_CV" * 0.95; END_IF;
END_REGION

REGION Network 12: If PID enabled, add ambient base to target
   RUNG wire#powerrail
      Contact( "PID_Bon4_Enable" )
      { S7_Templates := "SrcType := Real"; S7_GenerateENO := "TRUE" } Add(in1 := "TT3219_Bon4_Target", in2 := 25.0, out => "TT3219_Bon4_Target")
   END_RUNG
   // the same network as SCL:
   IF "PID_Bon4_Enable" THEN "TT3219_Bon4_Target" := "TT3219_Bon4_Target" + 25.0; END_IF;
END_REGION

REGION Network 13: If PID disabled, set target to ambient
   RUNG wire#powerrail
      I_Contact( "PID_Bon4_Enable" )
      { S7_GenerateENO := "TRUE" } Move(in := 25.0, out1 => "TT3219_Bon4_Target")
   END_RUNG
   // the same network as SCL:
   IF NOT "PID_Bon4_Enable" THEN "TT3219_Bon4_Target" := 25.0; END_IF;
END_REGION

REGION Network 14: Calculate memory term: Pure * 0.995
   RUNG wire#powerrail
      { S7_Templates := "SrcType := Real"; S7_GenerateENO := "TRUE" } Mul(in1 := "TT3219_Bon4_Sim_Pure", in2 := 0.995, out => "PID_Bon4_Temp_Val_1")
   END_RUNG
   // the same network as SCL:
   "PID_Bon4_Temp_Val_1" := "TT3219_Bon4_Sim_Pure" * 0.995;
END_REGION

REGION Network 15: Calculate target term: Target * 0.005
   RUNG wire#powerrail
      { S7_Templates := "SrcType := Real"; S7_GenerateENO := "TRUE" } Mul(in1 := "TT3219_Bon4_Target", in2 := 0.005, out => "PID_Bon4_Temp_Val_2")
   END_RUNG
   // the same network as SCL:
   "PID_Bon4_Temp_Val_2" := "TT3219_Bon4_Target" * 0.005;
END_REGION

REGION Network 16: Combine terms: Pure = Pure_prev * 0.995 + Target * 0.005
   RUNG wire#powerrail
      { S7_Templates := "SrcType := Real"; S7_GenerateENO := "TRUE" } Add(in1 := "PID_Bon4_Temp_Val_1", in2 := "PID_Bon4_Temp_Val_2", out => "TT3219_Bon4_Sim_Pure")
   END_RUNG
   // the same network as SCL:
   "TT3219_Bon4_Sim_Pure" := "PID_Bon4_Temp_Val_1" + "PID_Bon4_Temp_Val_2";
END_REGION

REGION Network 17: Increment simulation counter
   RUNG wire#powerrail
      { S7_Templates := "SrcType := Real"; S7_GenerateENO := "TRUE" } Add(in1 := "PID_Bon4_Sim_Counter", in2 := 1.0, out => "PID_Bon4_Sim_Counter")
   END_RUNG
   // the same network as SCL:
   "PID_Bon4_Sim_Counter" := "PID_Bon4_Sim_Counter" + 1.0;
END_REGION

REGION Network 18: Reset simulation counter at 1000
